	gripTime			   : TIME := T#250MS;                          // Време за ход на грипера
	gripTimeOut            : TIME := T#2S;                             // Време за отваряне/затваряне на гриперите
	insertTimeOut          : TIME := T#3S;                             // Време за движене нагоре/надолу на inserter 
    driveMoveTimeOut	   : TIME := T#4S;                             // Време за ход на мотора
	driveHomeTimeOut       : TIME := T#10S;                            // Време за home на мотора
	camTimeOut             : TIME := T#2S; 							   // Време за 1 снимка от камерата
	driveEnTime            : TIME := T#1S;                             // Време за ресет на инвертора на мотора
	drivePosTime           : TIME := T#100MS;                          // Време за задаване на задание за позициониране	

END_VAR


drivesControl();          // Упр. на ЛинМот мотора 

setStateVars(ioImage, activeState);


CASE activeState OF


//  *** Start Up
//  Старт на станцията след подаване на захр.	

	inserterLoadStates.stStartUp:
		setDisplayState(inserterLoadDisplayStates.dStStartUp);
		Stations.insertLoadDrive.DoEnable   := FALSE;
		Stations.insertLoadDrive.DoMove     := FALSE;	
		Stations.insertLoadDrive.DoHome     := FALSE;					   						   
		nextState(inserterLoadStates.stPowerUp);

//  *** Power Up - Start
//  Инициализация след подaване на захранване

	inserterLoadStates.stPowerUp:
		IF io.getSR(ioImage.xGrip_close, ioImage.xGrip_open) THEN
			setError(inserterLoadStates.stErrInitSensor);
		END_IF
		nextState(inserterLoadStates.stInit);

//  *** Init 
//  Инициализация на станцията
	
	inserterLoadStates.stInit:
	
		depWait(globalDeps.depILoadInitDone);		
		
		IF NOT resetDone THEN
			nextState(inserterLoadStates.stResetStart);
		END_IF
		
		IF prepareStart THEN
			nextState(inserterLoadStates.stPrepareStart);
		END_IF
		
		IF loadStart THEN
			nextState(inserterLoadStates.stLoadStart);
		END_IF		
		
		IF rotStart THEN
			nextState(inserterLoadStates.stRotStart);
		END_IF

		IF posStart THEN
			nextState(inserterLoadStates.stPosStart);
		END_IF

		IF insertStart THEN
			nextState(inserterLoadStates.stInsertStart);		
		END_IF	

		IF releaseStart THEN
			nextState(inserterLoadStates.stReleaseStart);
		END_IF	

		IF syncStart THEN
			nextState(inserterLoadStates.stSyncIndexStart);
		END_IF		
			
		nextState(inserterLoadStates.stInitDone);
		
// *** Init Done

	inserterLoadStates.stInitDone:
		nextState(inserterLoadStates.stReady);
	
// *** Ready

	inserterLoadStates.stReady:	
		setDisplayState(inserterLoadDisplayStates.dStStandBy);	
		IF Global.purgeDoneIL THEN
			resetDone          := FALSE;		
			Global.purgeDoneIL := FALSE;
		END_IF
		depNextState(Stations.machineStBase, GlobalDeps.depMachineStopping,  inserterLoadStates.stInserterLoadStopped);
		depNextState(Stations.machineStBase, GlobalDeps.depMachineStop,      inserterLoadStates.stInserterLoadStopped);	
		depWait(globalDeps.depILoadWaitIndex);
		nextState(inserterLoadStates.stPrepareStart);

// *** Inserter is Stopped

	inserterLoadStates.stInserterLoadStopped:
		setDisplayState(inserterLoadDisplayStates.dStStationIsStopped);	
		depWait(globalDeps.depILoadStop);
		depNextState(stations.machineStBase, GlobalDeps.depMachineAuto,       inserterLoadStates.stReady);
	    depNextState(Stations.machineStBase, GlobalDeps.depMachinePurgeStart, inserterLoadStates.stReady);			
		Stations.insertLoadDrive.DoEnable   := FALSE;
		Stations.insertLoadDrive.DoMove     := FALSE;	
		Stations.insertLoadDrive.DoHome     := FALSE;		

// *** Reset - Start
// Ресетиране на inserter

	inserterLoadStates.stResetStart:
		setDisplayState(inserterLoadDisplayStates.dStStationIsReseting);		
		resetDone := FALSE;		
		nextState(inserterLoadStates.stResetSyncRobot);
		
// *** Reset - Robot Sync
// Робота трябва да е на безопастно растояние

	inserterLoadStates.stResetSyncRobot:
		IF NOT GLobal.robotSafe THEN	
			depWait(globalDeps.depILoadWaitRobotReady);
			nextState(inserterLoadStates.stResetGripOpen);	
		ELSE
			nextState(inserterLoadStates.stResetGripOpen);	
		END_IF			

// *** Reset - Grip Open
// Отваряне на грипера

	inserterLoadStates.stResetGripOpen:
		io.setSR(ioImage.yGrip_open, ioImage.yGrip_close);
		nextState(inserterLoadStates.stResetGripCheck);	

// *** Reset - Grip Check
// Проверка дали грипера се е отворил
// Движение на гора на инсертъра

	inserterLoadStates.stResetGripCheck:		
 		IF io.getSR(ioImage.xGrip_open, ioImage.xGrip_close) THEN
			io.setSR(ioImage.yInsert_up, ioImage.yInsert_down);
			nextState(inserterLoadStates.stResetMoveUpCheck);	
		END_IF
		timeOutError(gripTimeOut, inserterLoadStates.stErrGripNotOpen);
		
// *** Reset - Move Up Check
// Проверка дали инсертъра е горе

	inserterLoadStates.stResetMoveUpCheck:		
		IF io.getSR(ioImage.xInsert_up, ioImage.xInsert_down) THEN
			nextState(inserterLoadStates.stResetLimitsCalc);			
		END_IF
		timeOutError(insertTimeOut, inserterLoadStates.stErrInsertNotUp);	
			
// *** Reset - Limit Check
// В зависимост от избраният модел на продукт се зараждат настойки в инвертора на мотора

	inserterLoadStates.stResetLimitsCalc:
			
		initRotPos    := Stations.insertLoadSetting.rotParams[Global.recipe].initRot;
		camRotPos     := Stations.insertLoadSetting.rotParams[Global.recipe].camRot;
		cwRotPos      := Stations.insertLoadSetting.rotParams[Global.recipe].cwRot;
		ccwRotPos     := Stations.insertLoadSetting.rotParams[Global.recipe].ccwRot;
		
		IF Stations.insertLoadDrive.Error THEN
			Stations.insertLoadDrive.DoReset  := TRUE;
		ELSE
			Stations.insertLoadDrive.DoReset  := FALSE;
			Stations.insertLoadDrive.DoEnable := TRUE;
			IF stateDelay(driveEnTime) THEN
				nextState(inserterLoadStates.stResetDriveHome);
			END_IF
		END_IF
		timeOutError(driveEnTime*2, inserterLoadStates.stErrDriveErr);
		
// *** Reset - Drive Home
// Рефериране на мотора

	inserterLoadStates.stResetDriveHome:		
		IF Stations.insertLoadDrive.Enabled AND NOT Stations.insertLoadDrive.Error THEN	
			Stations.insertLoadDrive.DoHome := TRUE;
			IF stateDelay(driveEnTime) THEN
				nextState(inserterLoadStates.stResetDriveCheck1);	
			END_IF
		ELSE
			setError(inserterLoadStates.stErrDriveErr);
	   END_IF	
		
// *** Reset - Drive Check
// Проверка дали реферирането на мотора е завършено

	inserterLoadStates.stResetDriveCheck1:		
		IF Stations.insertLoadDrive.Refferenced AND NOT Stations.insertLoadDrive.Error THEN
			Stations.insertLoadDrive.DoHome := FALSE;
			nextState(inserterLoadStates.stResetDriveMove);	
		END_IF
		timeOutError(driveHomeTimeOut, inserterLoadStates.stErrDriveHome);	

// *** Reset - Drive Move
// Ротатора застава на начална позиция

	inserterLoadStates.stResetDriveMove:
		IF Stations.insertLoadDrive.Enabled AND NOT Stations.insertLoadDrive.Error THEN	
			Stations.insertLoadDrive.TargetVelocity      := Stations.insertLoadSetting.axisWorkSpeed;
			Stations.insertLoadDrive.TargetAcceleration  := Stations.insertLoadSetting.axisAcc;
			Stations.insertLoadDrive.TargetPrecision     := Stations.insertLoadSetting.axisPres;
			Stations.insertLoadDrive.TargetPosition      := initRotPos;
		    Stations.insertLoadDrive.DoMove              := TRUE;
			IF stateDelay(driveEnTime) THEN			
				nextState(inserterLoadStates.stResetDriveCheck2);	
			END_IF
		ELSE
			setError(inserterLoadStates.stErrDriveErr);
	   END_IF	
	   
// *** Reset - Drive Check2
// Проверка дали реферирането на мотора е завършено

	inserterLoadStates.stResetDriveCheck2:		
		IF Stations.insertLoadDrive.TargetReached AND NOT Stations.insertLoadDrive.Error THEN
			Stations.insertLoadDrive.DoMove := FALSE;
			nextState(inserterLoadStates.stResetDone);	
		ELSIF NOT Stations.insertLoadDrive.TargetReached AND Stations.insertLoadDrive.Error THEN
			setError(inserterLoadStates.stErrDriveErr);
		END_IF	
		timeOutError(driveMoveTimeOut, inserterLoadStates.stErrDriveTimeOut);	

// *** Reset - Done

	inserterLoadStates.stResetDone:		
		resetDone := TRUE;
	    nextState(inserterLoadStates.stReady);			
		
// *** Prepare - Start
// Индекс масата е завършила ходата си - чака се робота да донесе сензор

	inserterLoadStates.stPrepareStart:
	   setDisplayState(inserterLoadDisplayStates.dStWorking);
	   prepareStart := TRUE;
	   nextState(inserterLoadStates.stPrepareNestCheck);	   
	   
// *** Prepare - Nest Check
// Ако в масата има зареден сенсор - станцията преключва работа
// Иначе дава сигнал на робота, че очаква от него да донесе сензор

	inserterLoadStates.stPrepareNestCheck:	   
		IF NOT io.getX(ioImage.xNest) AND NOT Global.purgeActive THEN
 	       nextState(inserterLoadStates.stPrepareRobotWait);  
        ELSE
	        prepareStart := FALSE;
 	        nextState(inserterLoadStates.stSyncIndexStart);  			
        END_IF	
	  
// *** Prepare - Robot Wait
// Изчаква робота да донесе сензор 

	inserterLoadStates.stPrepareRobotWait:		
		depSignal(globalDeps.depILoadSignalForLoad);
		depNextState(Stations.roboStBase, globalDeps.depRoboILoadOnPos, inserterLoadStates.stPrepareDone);
	
// *** Prepare - Done 

	inserterLoadStates.stPrepareDone:		
		prepareStart    := FALSE;
		nextState(inserterLoadStates.stLoadStart);
		
// *** Load - Start
// Сензора трябва да се прехвърли от робота в грипера на инсъртъра

	inserterLoadStates.stLoadStart:			
		loadStart   := TRUE;
		io.setSR(ioImage.yGrip_close, ioImage.yGrip_open);
		IF stateDelay(gripTime) THEN
			nextState(inserterLoadStates.stLoadGripCheck);	
		END_IF
	
// *** Load - Gripper Check
// Проверява се дали се е затворил грипера на инсъртъра

	inserterLoadStates.stLoadGripCheck:		
		IF io.getSR(ioImage.xGrip_close, ioImage.xGrip_open) THEN
			nextState(inserterLoadStates.stLoadRobotSync);	
		END_IF	
		timeOutError(gripTimeOut, inserterLoadStates.stErrGripNotClose);		
		
// *** Load - Robo Sync
// Дава се сигнал робота да си отвори грипера

	inserterLoadStates.stLoadRobotSync:			
		depWait(globalDeps.depRoboGripOpen);
		depNextState(Stations.roboStBase, GlobalDeps.depILoadRobotBack, inserterLoadStates.stLoadDone);

// *** Load - Done

	inserterLoadStates.stLoadDone:			
		loadStart  := FALSE;
		nextState(inserterLoadStates.stRotStart);		

// *** Rot - Start
// Започва ротиране на сензора, за да може да бъде сниман

	inserterLoadStates.stRotStart:	
		rotStart    := TRUE;
		io.setSR(ioImage.yGrip_close, ioImage.yGrip_open);
		nextState(inserterLoadStates.stRotGripCheck);

// *** Rot - Grip Check
// Ако е затворен грипера, пуска мотора 

	inserterLoadStates.stRotGripCheck:
		IF io.getSR(ioImage.xGrip_close, ioImage.xGrip_open) THEN
			IF Stations.insertLoadDrive.Enabled AND NOT Stations.insertLoadDrive.Error THEN
				nextState(inserterLoadStates.stRotDriveMove);	
			ELSE
			    nextState(inserterLoadStates.stRotDriveOn);			
			END_IF
		END_IF	
		timeOutError(gripTimeOut, inserterLoadStates.stErrGripNotClose);
		
// *** Rot - Drive On
// Ако е затворен грипера, пуска мотора 

	inserterLoadStates.stRotDriveOn:
		IF Stations.insertLoadDrive.Error THEN
			Stations.insertLoadDrive.DoReset  := TRUE;
		ELSE
			Stations.insertLoadDrive.DoReset  := FALSE;
			Stations.insertLoadDrive.DoEnable := TRUE;
			IF stateDelay(driveEnTime) THEN
				nextState(inserterLoadStates.stRotDriveMove);
			END_IF
		END_IF
		timeOutError(driveEnTime*2, inserterLoadStates.stErrDriveErr);

// *** Rot - Drive Move
// Завърта мотора на поз. за снимане

	inserterLoadStates.stRotDriveMove:
		IF Stations.insertLoadDrive.Enabled AND NOT Stations.insertLoadDrive.Error THEN	
			Stations.insertLoadDrive.TargetVelocity      := Stations.insertLoadSetting.axisWorkSpeed;
			Stations.insertLoadDrive.TargetAcceleration  := Stations.insertLoadSetting.axisAcc;
			Stations.insertLoadDrive.TargetPrecision     := Stations.insertLoadSetting.axisPres;
			Stations.insertLoadDrive.TargetPosition      := camRotPos;
		    Stations.insertLoadDrive.DoMove              := TRUE;	
			IF stateDelay(driveEnTime) THEN		
				nextState(inserterLoadStates.stRotDriveCheck);	
			END_IF
		ELSE
			setError(inserterLoadStates.stErrDriveErr);
	   END_IF	

// *** Rot - Drive Check
// Проверка дали мотора си е завършил хода

	inserterLoadStates.stRotDriveCheck:
		IF Stations.insertLoadDrive.TargetReached AND NOT Stations.insertLoadDrive.Error THEN
			Stations.insertLoadDrive.DoMove := FALSE;
			io.setY(ioImage.yFlashLight);
			nextState(inserterLoadStates.stRotCamShot);	
		ELSIF NOT Stations.insertLoadDrive.TargetReached AND Stations.insertLoadDrive.Error THEN
			setError(inserterLoadStates.stErrDriveErr);
		END_IF	
		timeOutError(driveMoveTimeOut, inserterLoadStates.stErrDriveTimeOut);

// *** Rot - Cam Shot
// Прави се снимка на сензора

	inserterLoadStates.stRotCamShot:
		Stations.insertLoadData := Global.recipe;
		nextState(inserterLoadStates.stRotCamCheck);

// *** Rot - Cam Check
// Проверява се дали има успешна снимка и върнат резултат

	inserterLoadStates.stRotCamCheck:
		IF Stations.insertLoadData = dataRequestCam.done THEN 
			io.rstY(ioImage.yFlashLight);
			
			IF TagsHMI.camResult <> camResult.null THEN
				
				CASE TagsHMI.camResult OF 
						camResult.turnCCW : workRotPos := ccwRotPos;
						camResult.turnCW  : workRotPos := cwRotPos;
				END_CASE
				nextState(inserterLoadStates.stRotDone);
				
			ELSE
				setError(inserterLoadStates.stErrCamBadResult);				
			END_IF
		
		ELSIF Stations.insertLoadData = dataRequestCam.error THEN
			setError(inserterLoadStates.stErrCamErr);			
		END_IF
		timeOutError(camTimeOut, inserterLoadStates.stErrCamTimeout);		
		
// *** Rot - Done

	inserterLoadStates.stRotDone:		
		rotStart   := FALSE;
		nextState(inserterLoadStates.stPosStart);		
		
// *** Pos  - Start
// Трябва да се завърти сензора на базата на резултата от камерата

	inserterLoadStates.stPosStart:		
		posStart   := TRUE;
		io.setSR(ioImage.yGrip_close, ioImage.yGrip_open);
		nextState(inserterLoadStates.stPosGripCheck);		
			
// *** Pos - Grip Check

	inserterLoadStates.stPosGripCheck:
		IF io.getSR(ioImage.xGrip_close, ioImage.xGrip_open) THEN
			IF Stations.insertLoadDrive.Enabled AND NOT Stations.insertLoadDrive.Error THEN
				nextState(inserterLoadStates.stPosDriveMove);	
			ELSE
			    nextState(inserterLoadStates.stPosDriveOn);			
			END_IF
		END_IF	
		timeOutError(gripTimeOut, inserterLoadStates.stErrGripNotClose);	
		
// *** Pos - Drive On
// Ако е затворен грипера, пуска мотора 

	inserterLoadStates.stPosDriveOn:
		IF Stations.insertLoadDrive.Error THEN
			Stations.insertLoadDrive.DoReset  := TRUE;
		ELSE
			Stations.insertLoadDrive.DoReset  := FALSE;
			Stations.insertLoadDrive.DoEnable := TRUE;
			IF stateDelay(driveEnTime) THEN
				nextState(inserterLoadStates.stPosDriveMove);
			END_IF
		END_IF
		timeOutError(driveEnTime*2, inserterLoadStates.stErrDriveErr);	
		
// *** Pos - Drive Move
// Завърта мотора 

	inserterLoadStates.stPosDriveMove:
		IF Stations.insertLoadDrive.Enabled AND NOT Stations.insertLoadDrive.Error THEN	
			Stations.insertLoadDrive.TargetVelocity      := Stations.insertLoadSetting.axisWorkSpeed;
			Stations.insertLoadDrive.TargetAcceleration  := Stations.insertLoadSetting.axisAcc;
			Stations.insertLoadDrive.TargetPrecision     := Stations.insertLoadSetting.axisPres;
			Stations.insertLoadDrive.TargetPosition      := workRotPos;
		    Stations.insertLoadDrive.DoMove              := TRUE;
			IF stateDelay(driveEnTime) THEN			
				nextState(inserterLoadStates.stPosDriveCheck);	
			END_IF
		ELSE
			setError(inserterLoadStates.stErrDriveErr);
	   END_IF	
		
// *** Pos - Drive Check
// Проверка дали мотора си е завършил хода

	inserterLoadStates.stPosDriveCheck:
		IF Stations.insertLoadDrive.TargetReached AND NOT Stations.insertLoadDrive.Error THEN
			Stations.insertLoadDrive.DoMove := FALSE;
			nextState(inserterLoadStates.stPosDone);	
		ELSIF NOT Stations.insertLoadDrive.TargetReached AND Stations.insertLoadDrive.Error THEN
			setError(inserterLoadStates.stErrDriveErr);
		END_IF	
		timeOutError(driveMoveTimeOut, inserterLoadStates.stErrDriveTimeOut);			   
	   
// *** Pos - Done

	inserterLoadStates.stPosDone:
		posStart   := FALSE;
		nextState(inserterLoadStates.stInsertStart);	  

// *** Insert - Start
// Поставя сензора на в гнездото на индекс масата

	inserterLoadStates.stInsertStart:
		insertStart := TRUE;
		io.setSR(ioImage.yGrip_close, ioImage.yGrip_open);
		nextState(inserterLoadStates.stInsertGripCheck);	

// *** Insert - Grip Check
// Проверява се дали грипера е затворен

	inserterLoadStates.stInsertGripCheck:
		IF io.getSR(ioImage.xGrip_close, ioImage.xGrip_open) THEN
			nextState(inserterLoadStates.stInsertNestCheck);		
		END_IF
		timeOutError(gripTimeOut, inserterLoadStates.stErrGripNotClose);
		
// *** Insert - Nest Check
// Сензор се поставя само ако на масата няма

	inserterLoadStates.stInsertNestCheck:
		IF NOT io.getX(ioImage.xNest) THEN
			io.setSR(ioImage.yInsert_down, ioImage.yInsert_up);
			nextState(inserterLoadStates.stInsertMoveDownCheck);			
		ELSE
			setError(inserterLoadStates.stErrInitSensor);
		END_IF
		
// *** Insert - Insert Move Down Check
// Проверява се дали е инсъртъра е долу

	inserterLoadStates.stInsertMoveDownCheck:		
		IF io.getSR(ioImage.xInsert_down, ioImage.xInsert_up) THEN
			nextState(inserterLoadStates.stInsetDone);			
		END_IF	
		timeOutError(insertTimeOut, inserterLoadStates.stErrInsertNotDown);

// *** Insert - Done

	inserterLoadStates.stInsetDone:	 
		insertStart := FALSE;
		nextState(inserterLoadStates.stReleaseStart);		
	   
// *** Release - Start
// Оставяне на сензора в гнездота и връщата в начална поз.

	inserterLoadStates.stReleaseStart:	   
		releaseStart := TRUE;
		io.setSR(ioImage.yGrip_open, ioImage.yGrip_close);
		nextState(inserterLoadStates.stReleaseGripCheck);	

// *** Release - Grip Check
// Проверка дали грипера се е отворил

	inserterLoadStates.stReleaseGripCheck:	   
		IF io.getSR(ioImage.xGrip_open, ioImage.xGrip_close) THEN
			io.setSR(ioImage.yInsert_up, ioImage.yInsert_down);
			nextState(inserterLoadStates.stReleaseMoveUpCheck);			
		END_IF	
		timeOutError(gripTimeOut, inserterLoadStates.stErrGripNotOpen);				   
	
// *** Release - Move Up Check
// Проверка дали инсъртъра е горе

	inserterLoadStates.stReleaseMoveUpCheck:
		IF io.getSR(ioImage.xInsert_up, ioImage.xInsert_down) THEN
			IF Stations.insertLoadDrive.Enabled AND NOT Stations.insertLoadDrive.Error THEN
				nextState(inserterLoadStates.stReleaseDriveMove);	
			ELSE
			    nextState(inserterLoadStates.stReleaseDriveOn);			
			END_IF			
		END_IF
		timeOutError(insertTimeOut, inserterLoadStates.stErrInsertNotUp);	

// *** Release - Drive On
// Ако инсъртъра е горе , пуска мотора 

	inserterLoadStates.stReleaseDriveOn:
		IF Stations.insertLoadDrive.Error THEN
			Stations.insertLoadDrive.DoReset  := TRUE;
		ELSE
			Stations.insertLoadDrive.DoReset  := FALSE;
			Stations.insertLoadDrive.DoEnable := TRUE;
			IF stateDelay(driveEnTime) THEN
				nextState(inserterLoadStates.stReleaseDriveMove);
			END_IF
		END_IF
		timeOutError(driveEnTime*2, inserterLoadStates.stErrDriveErr);	
		
// *** Release - Drive Move
// Завърта мотора 

	inserterLoadStates.stReleaseDriveMove:
		IF Stations.insertLoadDrive.Enabled AND NOT Stations.insertLoadDrive.Error THEN	
			Stations.insertLoadDrive.TargetVelocity      := Stations.insertLoadSetting.axisWorkSpeed;
			Stations.insertLoadDrive.TargetAcceleration  := Stations.insertLoadSetting.axisAcc;
			Stations.insertLoadDrive.TargetPrecision     := Stations.insertLoadSetting.axisPres;
			Stations.insertLoadDrive.TargetPosition      := initRotPos;
		    Stations.insertLoadDrive.DoMove              := TRUE;
			IF stateDelay(driveEnTime) THEN			
				nextState(inserterLoadStates.stReleaseDriveCheck);	
			END_IF
		ELSE
			setError(inserterLoadStates.stErrDriveErr);
	   END_IF	
		
// *** Release - Drive Check
// Проверка дали мотора си е завършил хода

	inserterLoadStates.stReleaseDriveCheck:
		IF Stations.insertLoadDrive.TargetReached AND NOT Stations.insertLoadDrive.Error THEN
			Stations.insertLoadDrive.DoMove := FALSE;
			nextState(inserterLoadStates.stReleaseDone);	
		ELSIF NOT Stations.insertLoadDrive.TargetReached AND Stations.insertLoadDrive.Error THEN
			setError(inserterLoadStates.stErrDriveErr);
		END_IF	
		timeOutError(driveMoveTimeOut, inserterLoadStates.stErrDriveTimeOut);  
	   
// *** Release - Done

	inserterLoadStates.stReleaseDone:	
        setDisplayState(inserterLoadDisplayStates.dStStationReady);	
		releaseStart  := FALSE;
		nextState(inserterLoadStates.stSyncIndexStart);

// *** Sync Index - Start
// Дава се разрешение да се завърти индекс масата

	inserterLoadStates.stSyncIndexStart:
		syncStart := TRUE;		
		depWait(globalDeps.depILoadDone);	
		depNextState(Stations.incCommStBase, globalDeps.depIncCycleDone, inserterLoadStates.stSyncIndexDone); 

// *** Sync Index - Done

	inserterLoadStates.stSyncIndexDone:
		syncStart := FALSE;
		nextState(inserterLoadStates.stReady);   
	        
// *** Step Block State
// В този state се влиза винаги след изпълняването на една стъпка при стъпков режим
	inserterLoadStates.stStepBlock:
        setDisplayState(inserterLoadDisplayStates.dStWaitForNextStep);	
		
// *** Station Stop
// Станцията е била изключена 
 
	inserterLoadStates.stStop: 	
		Stations.insertLoadDrive.DoEnable   := FALSE;
		Stations.insertLoadDrive.DoMove     := FALSE;	
	    resetDone			                := FALSE; 						   
	    prepareStart                        := FALSE; 						   
	    loadStart                           := FALSE; 						   
	    rotStart                            := FALSE; 						   
	    posStart                            := FALSE; 						   
	    insertStart                         := FALSE;							  
	    releaseStart                        := FALSE; 						   
	    syncStart			                := FALSE; 

// *** ERROR - Grip Not Open
// Грипера не се е отворил на време

	inserterLoadStates.stErrGripNotOpen:
		setDisplayState(inserterLoadDisplayStates.dStGripperDidNotOpen); 

// *** ERROR - Grip Not Close
// Грипера не се е затворил на време

	inserterLoadStates.stErrGripNotClose:
		setDisplayState(inserterLoadDisplayStates.dStGripperDidNotClose);
		
// *** ERROR - Inserter Not Down
// Inserter не е стинглал долна позиция на време

	inserterLoadStates.stErrInsertNotDown:
		setDisplayState(inserterLoadDisplayStates.dStInserterDidNotMoveDown);		
		
// *** ERROR - Inserter Not Up
// Inserter не е стинглал горна позиция на време

	inserterLoadStates.stErrInsertNotUp:
		setDisplayState(inserterLoadDisplayStates.dStInserterDidNotMoveUp);		
		
// *** ERROR - Drive Homming TimeOut
// ЛинМот мотора не е могъл да се homming както трябва

	inserterLoadStates.stErrDriveHome:
		setDisplayState(inserterLoadDisplayStates.dStDriveDidNotHome);
		Stations.insertLoadDrive.DoEnable   := FALSE;
		Stations.insertLoadDrive.DoMove     := FALSE;	
		Stations.insertLoadDrive.DoHome     := FALSE;	
		
// *** ERROR - Drive Homming TimeOut
// ЛинМот инвертора е върнал грешка

	inserterLoadStates.stErrDriveErr:
		setDisplayState(inserterLoadDisplayStates.dStDriveError);	
		Stations.insertLoadDrive.DoEnable   := FALSE;
		Stations.insertLoadDrive.DoMove     := FALSE;		
		
// *** ERROR - Drive Move TimeOut
// ЛинМот мотора не е завършил движението си навреме

	inserterLoadStates.stErrDriveTimeOut:
		setDisplayState(inserterLoadDisplayStates.dStDriveTimeOutMove);	
		Stations.insertLoadDrive.DoEnable   := FALSE;
		Stations.insertLoadDrive.DoMove     := FALSE;		
		
// *** ERROR - Camera Timeout
// Камерата се е забавила твърде мн. с връщането на резултат

	inserterLoadStates.stErrCamTimeout:
		setDisplayState(inserterLoadDisplayStates.dStCameraTimeOut);
		
// *** ERROR - Camera Error
// Камерата се е забавила твърде мн. с връщането на резултат

	inserterLoadStates.stErrCamErr:
		setDisplayState(inserterLoadDisplayStates.dStCameraError);
		
// *** ERROR - Camera Error
// Камерата е върнала грешен резултат

	inserterLoadStates.stErrCamBadResult:
		setDisplayState(inserterLoadDisplayStates.dStCameraBadResult);	
		
	
// *** ERROR - Init sensor 
// При старт на машаината не може да има захванат от грипера сензор

	inserterLoadStates.stErrInitSensor:	
		setDisplayState(inserterLoadDisplayStates.dStInitSensorGripError);	
		
// *** EMG Stop
// Аварийно спиране при натискане на гъба или отваряне на врата

	inserterLoadStates.stEMG:		
		Stations.insertLoadDrive.DoEnable   := FALSE;
		Stations.insertLoadDrive.DoMove     := FALSE;	
		Stations.insertLoadDrive.DoHome     := FALSE;
		nextState(inserterLoadStates.stInit);		


END_CASE

ACTION drivesControl:


axisLinMot       ( TargetPosition 		   := Stations.insertLoadDrive.TargetPosition,
				   TargetVelocity 		   := Stations.insertLoadDrive.TargetVelocity,
				   TargetAcceleration	   := Stations.insertLoadDrive.TargetAcceleration,
				   TargetDeceleration	   := Stations.insertLoadDrive.TargetAcceleration,
				   TargetPrecision 		   := Stations.insertLoadDrive.TargetPrecision,			
				   IsAbsolute 			   := FALSE,
	               OperationMode		   := Stations.insertLoadDrive.OperationMode,     				
	               Enabled 				   => Stations.insertLoadDrive.Enabled,
	               Error 				   => Stations.insertLoadDrive.Error,
	               ErrorID 				   => Stations.insertLoadDrive.ErrorID,
	               Refferenced 			   => Stations.insertLoadDrive.Refferenced,
	               Moving 				   => Stations.insertLoadDrive.Moving,
	               CurrentPosition 		   => Stations.insertLoadDrive.CurrentPosition,
	               CurrentVelocity		   => Stations.insertLoadDrive.CurrentVelocity,             				
				   Axis					   := Stations.insertLoadAxis,
		           DoServoOn 			   := Stations.insertLoadDrive.DoEnable, 
	               DoHome 				   := Stations.insertLoadDrive.DoHome, 
	               DoMove 				   := Stations.insertLoadDrive.DoMove, 
	               DoReset 				   := Stations.insertLoadDrive.DoReset, 
	               TargetReached 		   := Stations.insertLoadDrive.TargetReached, 
	               DoStop 				   := Stations.insertLoadDrive.DoStop);
END_ACTION

END_FUNCTION_BLOCK

// ---- POUs/Stations/insertUnloadStation.TcPOU
FUNCTION_BLOCK insertUnloadStation EXTENDS stateMachine
VAR_INPUT
	
	ioImage                : inserterUnloadImage;

END_VAR

VAR

	activeState            : inserterUnloadStates;	
	axisLinMot             : FB_ServoAxis_LinMot; 
	
	resetDone			   : BOOL := FALSE; 						   // Инсъртъра е ресетнат
	prepareStart           : BOOL := FALSE; 						   // Ако има сенсор в гнездото, завърта грипера 
	moveDownStart          : BOOL := FALSE; 						   // Слиза да вземе сензора
	unloadSensorStart      : BOOL := FALSE; 						   // Взима сензора и инсъртъра се вдига нагоре
	posStart               : BOOL := FALSE; 						   // Ротира грипера за взимане на сензора от робота
	releaseStart           : BOOL := FALSE; 						   // Подава сензора на робота
	syncRobot              : BOOL := false;                            // Робота е на безопастно място
	syncStart			   : BOOL := FALSE; 						   // Sync с индекс масата, че работа е завършена
	
	
	initRotPos			   : REAL; 									   // Начално завъртане
	workRotPos             : REAL;                                     // Завъртане за може робота да вземе сензора
	
	gripTime			   : TIME := T#250MS;                          // Време за ход на грипера                                     
	gripTimeOut            : TIME := T#2S;                             // Време за отваряне/затваряне на гриперите
	insertTimeOut          : TIME := T#3S;                             // Време за движене нагоре/надолу на inserter
    driveMoveTimeOut	   : TIME := T#4S;                             // Време за ход на мотора
	driveHomeTimeOut       : TIME := T#10S;                            // Време за home на мотора
	sensorTime             : TIME := T#250MS; 						   // Време за за реакция на лазерен сензор
	driveEnTime            : TIME := T#1S;                             // Време за ресет на инвертора на мотора
	drivePosTime           : TIME := T#100MS;                          // Време за задаване на задание за позициониране	

END_VAR


drivesControl();          // Упр. на ЛинМот мотора 

setStateVars(ioImage, activeState);

CASE activeState OF
	

//  *** Start Up
//  Старт на станцията след подаване на захр.	

	inserterUnloadStates.stStartUp:
		setDisplayState(inserterUnLoadDisplayStates.dStStartUp);
		Stations.insertUnLoadDrive.DoEnable   := FALSE;
		Stations.insertUnLoadDrive.DoMove     := FALSE;	
		Stations.insertUnLoadDrive.DoHome     := FALSE;					   						   
		nextState(inserterUnloadStates.stPowerUp);

//  *** Power Up - Start
//  Инициализация след подaване на захранване

	inserterUnloadStates.stPowerUp:
		IF io.getSR(ioImage.xGrip_close, ioImage.xGrip_open) THEN
			setError(inserterUnloadStates.stErrInitSensor);
		END_IF
		nextState(inserterUnloadStates.stInit);

//  *** Init 
//  Инициализация на станцията
	
	inserterUnloadStates.stInit:
	
		depWait(globalDeps.depULoadInitDone);	
		
		IF NOT resetDone THEN
			nextState(inserterUnloadStates.stResetStart);
		END_IF
		
		IF prepareStart THEN
			nextState(inserterUnloadStates.stPrepareStart);
		END_IF
		
		IF moveDownStart THEN
			nextState(inserterUnloadStates.stMoveDownStart);
		END_IF		
		
		IF unloadSensorStart THEN
			nextState(inserterUnloadStates.stUnloadSensorStart);
		END_IF

		IF posStart THEN
			nextState(inserterUnloadStates.stPosStart);
		END_IF

		IF releaseStart THEN
			nextState(inserterUnloadStates.stReleaseStart);
		END_IF	
		
		IF syncRobot THEN
			nextState(inserterUnloadStates.stReleaseDone);
		END_IF

		IF syncStart THEN
			nextState(inserterUnloadStates.stSyncIndexStart);
		END_IF		
			
		nextState(inserterUnloadStates.stInitDone);
		
// *** Init Done

	inserterUnloadStates.stInitDone:
		nextState(inserterUnloadStates.stReady);
	
// *** Ready

	inserterUnloadStates.stReady:	
		setDisplayState(inserterUnLoadDisplayStates.dStStandBy);	
		IF Global.purgeDoneIU THEN
			resetDone          := FALSE;		
			Global.purgeDoneIU := FALSE;
		END_IF
		depNextState(Stations.machineStBase, GlobalDeps.depMachineStopping,  inserterUnloadStates.stInserterUnloadStopped);
		depNextState(Stations.machineStBase, GlobalDeps.depMachineStop,      inserterUnloadStates.stInserterUnloadStopped);	
		depWait(globalDeps.depULoadWaitIndex);
		nextState(inserterUnloadStates.stPrepareStart);

// *** Inserter is Stopped

	inserterUnloadStates.stInserterUnloadStopped:
		setDisplayState(inserterUnLoadDisplayStates.dStStationIsStopped);
		depWait(globalDeps.depULoadStop);
		depNextState(stations.machineStBase, GlobalDeps.depMachineAuto,       inserterUnloadStates.stReady);
	    depNextState(Stations.machineStBase, GlobalDeps.depMachinePurgeStart, inserterUnloadStates.stReady);			
		Stations.insertUnLoadDrive.DoEnable   := FALSE;
		Stations.insertUnLoadDrive.DoMove     := FALSE;	
		Stations.insertUnLoadDrive.DoHome     := FALSE;

// *** Reset - Start
// Ресетиране на inserter

	inserterUnloadStates.stResetStart:
		setDisplayState(inserterUnLoadDisplayStates.dStStationIsReseting);	
		resetDone := FALSE;		
		nextState(inserterUnloadStates.stResetSyncRobot);
		
// *** Reset - Robot Sync
// Робота трябва да е на безопастно растояние

	inserterUnloadStates.stResetSyncRobot:
		IF NOT Global.robotSafe THEN	
			depWait(globalDeps.depULoadWaitRobotReady);
			nextState(inserterUnloadStates.stResetGripOpen);	
	    ELSE
			nextState(inserterUnloadStates.stResetGripOpen);
		END_IF		

// *** Reset - Grip Open
// Отваряне на грипера

	inserterUnloadStates.stResetGripOpen:
		io.setSR(ioImage.yGrip_open, ioImage.yGrip_close);
		nextState(inserterUnloadStates.stResetGripCheck);	

// *** Reset - Grip Check
// Проверка дали грипера се е отворил.
// Движение на гора на инсертъра

	inserterUnloadStates.stResetGripCheck:		
 		IF io.getSR(ioImage.xGrip_open, ioImage.xGrip_close) THEN
			io.setSR(ioImage.yInsert_up, ioImage.yInsert_down);
			nextState(inserterUnloadStates.stResetMoveUpCheck);	
		END_IF
		timeOutError(gripTimeOut, inserterUnloadStates.stErrGripNotOpen);
		
// *** Reset - Move Up Check
// Проверка дали инсертъра е горе

	inserterUnloadStates.stResetMoveUpCheck:		
		IF io.getSR(ioImage.xInsert_up, ioImage.xInsert_down) THEN
			nextState(inserterUnloadStates.stResetLimitsCalc);			
		END_IF
		timeOutError(insertTimeOut, inserterUnloadStates.stErrInsertNotUp);	
			
// *** Reset - Limit Check
// В зависимост от избраният модел на продукт се зараждат настойки в инвертора на мотора

	inserterUnloadStates.stResetLimitsCalc:
			
		initRotPos     := Stations.insertUnloadSetting.rotParams[Global.recipe].initRot;
		workRotPos     := Stations.insertUnloadSetting.rotParams[Global.recipe].workRot;

		
		IF Stations.insertUnLoadDrive.Error THEN
			Stations.insertUnLoadDrive.DoReset  := TRUE;
		ELSE
			Stations.insertUnLoadDrive.DoReset  := FALSE;
			Stations.insertUnLoadDrive.DoEnable := TRUE;
			IF stateDelay(driveEnTime) THEN
				nextState(inserterUnloadStates.stResetDriveHome);
			END_IF
		END_IF
		timeOutError(driveEnTime*2, inserterUnloadStates.stErrDriveErr);
		
// *** Reset - Drive Home
// Рефериране на мотора

	inserterUnloadStates.stResetDriveHome:		
		IF Stations.insertUnLoadDrive.Enabled AND NOT Stations.insertUnLoadDrive.Error THEN	
			Stations.insertUnLoadDrive.DoHome := TRUE;
			IF stateDelay(drivePosTime) THEN
				nextState(inserterUnloadStates.stResetDriveCheck);	
			END_IF	
		ELSE
			setError(inserterUnloadStates.stErrDriveErr);
	   END_IF	
		
// *** Reset - Drive Check
// Проверка дали реферирането на мотора е завършено

	inserterUnloadStates.stResetDriveCheck:		
		IF Stations.insertUnLoadDrive.Refferenced AND NOT Stations.insertUnLoadDrive.Error THEN
			Stations.insertUnLoadDrive.DoHome := FALSE;
			nextState(inserterUnloadStates.stResetDone);	
		END_IF
		timeOutError(driveHomeTimeOut, inserterUnloadStates.stErrDriveHome);	

// *** Reset - Done

	inserterUnloadStates.stResetDone:		
		resetDone := TRUE;
	    nextState(inserterUnloadStates.stReady);		
		
// *** Prepare - Start
// Индекс масата е завършила ходата си 

	inserterUnloadStates.stPrepareStart:
       setDisplayState(inserterUnLoadDisplayStates.dStWorking);	 
	   prepareStart := TRUE;
	   io.setSR(ioImage.yGrip_open, ioImage.yGrip_close);
	   io.setSR(ioImage.yInsert_up, ioImage.yInsert_down);
	   nextState(inserterUnloadStates.stPrepareGripCheck);		
		
// *** Prepare - Grip Check
// Инсертера трябва да е горе и грипера му да е отворен

	inserterUnloadStates.stPrepareGripCheck:		
		IF io.getSR(ioImage.xGrip_open, ioImage.xGrip_close) AND 
		   io.getSR(ioImage.xInsert_up, ioImage.xInsert_down) THEN
				nextState(inserterUnloadStates.stPrepareNestCheck);
		ELSE
			IF stateDelay(insertTimeOut) THEN
				IF NOT io.getSR(ioImage.xGrip_open, ioImage.xGrip_close) THEN
					setError(inserterUnloadStates.stErrGripNotOpen);
				ELSIF io.getSR(ioImage.xInsert_up, ioImage.xInsert_down) THEN
					setError(inserterUnloadStates.stErrInsertNotUp);
				END_IF
			END_IF
		END_IF	
				
// *** Prepare - Nest Check
// За да започне цикъла на станицята, трябва да има в сензор в гнездото
// и InC да е върнало, че този сензор е със статус GOOD

	inserterUnloadStates.stPrepareNestCheck:	
		IF stateDelay(sensorTime) THEN
			IF io.getX(ioImage.xNest) AND Global.sensorStatus THEN
				Global.sensorOnIUnload := TRUE; 			
				IF Stations.insertUnloadDrive.Enabled AND NOT Stations.insertUnloadDrive.Error THEN
					nextState(inserterUnloadStates.stPrepareDriveMove);
				ELSE
					nextState(inserterUnloadStates.stPrepareDriveOn);
				END_IF
			ELSIF io.getX(ioImage.xNest) XOR GLobal.sensorStatus THEN
				setError(inserterUnloadStates.stErrNestSensor);
			ELSE	
				prepareStart := FALSE;
				nextState(inserterUnloadStates.stSyncIndexStart);
			END_IF
		END_IF	

// *** Prepare - Drive On
// Захранване на мотора ако не е пуснат 

	inserterUnloadStates.stPrepareDriveOn:
		IF Stations.insertUnLoadDrive.Error THEN
			Stations.insertUnLoadDrive.DoReset  := TRUE;
		ELSE
			Stations.insertUnLoadDrive.DoReset  := FALSE;
			Stations.insertUnLoadDrive.DoEnable := TRUE;
			IF stateDelay(driveEnTime) THEN
				nextState(inserterUnloadStates.stPrepareDriveMove);
			END_IF
		END_IF
		timeOutError(driveEnTime*2, inserterUnloadStates.stErrDriveErr);

// *** Prepare - Drive Move
// Завърта мотора на поз. за изваждането на сензор

	inserterUnloadStates.stPrepareDriveMove:
		IF Stations.insertUnLoadDrive.Enabled AND NOT Stations.insertUnLoadDrive.Error THEN	
			Stations.insertUnLoadDrive.TargetVelocity      := Stations.insertUnLoadSetting.axisWorkSpeed;
			Stations.insertUnLoadDrive.TargetAcceleration  := Stations.insertUnLoadSetting.axisAcc;
			Stations.insertUnLoadDrive.TargetPrecision     := Stations.insertUnLoadSetting.axisPres;
			Stations.insertUnLoadDrive.TargetPosition      := initRotPos;
		    Stations.insertUnLoadDrive.DoMove              := TRUE;	
			IF stateDelay(drivePosTime) THEN		
				nextState(inserterUnloadStates.stPrepareDriveCheck);	
			END_IF	
		ELSE
			setError(inserterUnloadStates.stErrDriveErr);
	   END_IF	

// *** Prepare - Drive Check
// Проверка дали мотора си е завършил хода

	inserterUnloadStates.stPrepareDriveCheck:
		IF Stations.insertUnLoadDrive.TargetReached AND NOT Stations.insertUnLoadDrive.Error THEN
			Stations.insertUnLoadDrive.DoMove := FALSE;
			nextState(inserterUnloadStates.stPrepareDone);	
		ELSIF NOT Stations.insertUnLoadDrive.TargetReached AND Stations.insertUnLoadDrive.Error THEN
			setError(inserterUnloadStates.stErrDriveErr);
		END_IF	
		timeOutError(driveMoveTimeOut, inserterUnloadStates.stErrDriveTimeOut);

// *** Prepare - Done

	inserterUnloadStates.stPrepareDone:		
		prepareStart := FALSE;
	    nextState(inserterUnloadStates.stMoveDownStart);		
		
// *** Move Down  - Start
// Инсертера слиза надолу зада вземе сензор от гнездото на масата

	inserterUnloadStates.stMoveDownStart:	 
	   moveDownStart := TRUE;
	   io.setSR(ioImage.yGrip_open, ioImage.yGrip_close);
	   io.setSR(ioImage.yInsert_up, ioImage.yInsert_down);
	   nextState(inserterUnloadStates.stMoveDownGripCheck);	
		
// *** Move Down - Grip Check
// Инсертера трябва да е горе и грипера му да е отворен

	inserterUnloadStates.stMoveDownGripCheck:		
		IF io.getSR(ioImage.xGrip_open, ioImage.xGrip_close) AND 
		   io.getSR(ioImage.xInsert_up, ioImage.xInsert_down) THEN
		   		io.setSR(ioImage.yInsert_down, ioImage.yInsert_up);
				nextState(inserterUnloadStates.stMoveDownCheck);
		ELSE
			IF stateDelay(insertTimeOut) THEN
				IF NOT io.getSR(ioImage.xGrip_open, ioImage.xGrip_close) THEN
					setError(inserterUnloadStates.stErrGripNotOpen);
				ELSIF io.getSR(ioImage.xInsert_up, ioImage.xInsert_down) THEN
					setError(inserterUnloadStates.stErrInsertNotUp);
				END_IF
			END_IF
		END_IF			
		
// *** Move Down - Down Check
// Инсертера трябва да е долу

	inserterUnloadStates.stMoveDownCheck:		
		IF io.getSR(ioImage.xInsert_down, ioImage.xInsert_up) THEN
			nextState(inserterUnloadStates.stMoveDownDone);
		END_IF
		timeOutError(insertTimeOut, inserterUnloadStates.stErrInsertNotDown);	
		
// *** Move Down - Done

	inserterUnloadStates.stMoveDownDone:		
		moveDownStart := FALSE;
	    nextState(inserterUnloadStates.stUnloadSensorStart);		

// *** Unload Sensor - Start
// Грипера се затваря, захваща сензора и го изважда от гнездото на масата

	inserterUnloadStates.stUnloadSensorStart:	
		unloadSensorStart := TRUE;
		io.setSR(ioImage.yGrip_open, ioImage.yGrip_close);
		io.setSR(ioImage.yInsert_down, ioImage.yInsert_up);
	    nextState(inserterUnloadStates.stUnloadSensorGripCheck1);			

// *** Unload Sensor - Grip Check 1
// Проверка на гриперите

	inserterUnloadStates.stUnloadSensorGripCheck1:
		IF io.getSR(ioImage.xGrip_open, ioImage.xGrip_close) AND 
		   io.getSR(ioImage.xInsert_down, ioImage.xInsert_up) THEN
		   		io.setSR(ioImage.yGrip_close, ioImage.yGrip_open);
				nextState(inserterUnloadStates.stUnloadSensorGripCheck2);
		ELSE
			IF stateDelay(insertTimeOut) THEN
				IF NOT io.getSR(ioImage.xGrip_open, ioImage.xGrip_close) THEN
					setError(inserterUnloadStates.stErrGripNotOpen);
				ELSIF io.getSR(ioImage.xInsert_down, ioImage.xInsert_up) THEN
					setError(inserterUnloadStates.stErrInsertNotDown);
				END_IF
			END_IF
		END_IF	

// *** Unload Sensor - Grip Check 2
// Проверка  дали грипера се е затворил 

	inserterUnloadStates.stUnloadSensorGripCheck2:
		IF io.getSR(ioImage.xGrip_close, ioImage.xGrip_open) AND stateDelay(gripTime) THEN
			io.setSR(ioImage.yInsert_up, ioImage.yInsert_down);
			nextState(inserterUnloadStates.stUnloadSensorMoveCheck);
		END_IF	
		timeOutError(gripTimeOut, inserterUnloadStates.stErrGripNotClose);			
	
// *** Unload Sensor - Move Check
// Проверка  дали инсертера е горе

	inserterUnloadStates.stUnloadSensorMoveCheck:
		IF io.getSR(ioImage.xInsert_up, ioImage.xInsert_down) THEN
			nextState(inserterUnloadStates.stUnloadSensorDone);
		END_IF	
		timeOutError(insertTimeOut, inserterUnloadStates.stErrInsertNotUp);

// *** Unload Sensor - Done

	inserterUnloadStates.stUnloadSensorDone:		
		unloadSensorStart := FALSE;
	    nextState(inserterUnloadStates.stPosStart);
		
// *** Pos - Start
// Сензора трябва да се ротира, че да може да го хване робота

	inserterUnloadStates.stPosStart:
		posStart := TRUE;
		io.setSR(ioImage.yGrip_close, ioImage.yGrip_open);
		io.setSR(ioImage.yInsert_up, ioImage.yInsert_down);
		nextState(inserterUnloadStates.stPosGripCheck);

// *** Pos - Grip Check

	inserterUnloadStates.stPosGripCheck:		
		IF io.getSR(ioImage.xGrip_close, ioImage.xGrip_open) AND 
		   io.getSR(ioImage.xInsert_up, ioImage.xInsert_down) THEN
				IF Stations.insertUnloadDrive.Enabled AND NOT Stations.insertUnloadDrive.Error THEN
					nextState(inserterUnloadStates.stPosDriveMove);
				ELSE
					nextState(inserterUnloadStates.stPosDriveOn);
				END_IF
		ELSE
			IF stateDelay(insertTimeOut) THEN
				IF NOT io.getSR(ioImage.xGrip_close, ioImage.xGrip_open) THEN
					setError(inserterUnloadStates.stErrGripNotClose);
				ELSIF io.getSR(ioImage.xInsert_up, ioImage.xInsert_down) THEN
					setError(inserterUnloadStates.stErrInsertNotUp);
				END_IF
			END_IF
		END_IF			
		
// *** Pos - Drive On
// Захранване на мотора ако не е пуснат 

	inserterUnloadStates.stPosDriveOn:
		IF Stations.insertUnLoadDrive.Error THEN
			Stations.insertUnLoadDrive.DoReset  := TRUE;
		ELSE
			Stations.insertUnLoadDrive.DoReset  := FALSE;
			Stations.insertUnLoadDrive.DoEnable := TRUE;
			IF stateDelay(driveEnTime) THEN
				nextState(inserterUnloadStates.stPosDriveMove);
			END_IF
		END_IF
		timeOutError(driveEnTime*2, inserterUnloadStates.stErrDriveErr);

// *** Pos - Drive Move
// Завърта мотора на поз. за взимане на сензора от робота

	inserterUnloadStates.stPosDriveMove:
		IF Stations.insertUnLoadDrive.Enabled AND NOT Stations.insertUnLoadDrive.Error THEN	
			Stations.insertUnLoadDrive.TargetVelocity      := Stations.insertUnLoadSetting.axisWorkSpeed;
			Stations.insertUnLoadDrive.TargetAcceleration  := Stations.insertUnLoadSetting.axisAcc;
			Stations.insertUnLoadDrive.TargetPrecision     := Stations.insertUnLoadSetting.axisPres;
			Stations.insertUnLoadDrive.TargetPosition      := workRotPos;
		    Stations.insertUnLoadDrive.DoMove              := TRUE;	
			IF stateDelay(drivePosTime) THEN		
				nextState(inserterUnloadStates.stPosDriveCheck);
			END_IF	
		ELSE
			setError(inserterUnloadStates.stErrDriveErr);
	   END_IF	
		
// *** Pos - Drive Check
// Проверка дали мотора си е завършил хода

	inserterUnloadStates.stPosDriveCheck:
		IF Stations.insertUnLoadDrive.TargetReached AND NOT Stations.insertUnLoadDrive.Error THEN
			Stations.insertUnLoadDrive.DoMove := FALSE;
			nextState(inserterUnloadStates.stPosDone);	
		ELSIF NOT Stations.insertUnLoadDrive.TargetReached AND Stations.insertUnLoadDrive.Error THEN
			setError(inserterUnloadStates.stErrDriveErr);
		END_IF	
		timeOutError(driveMoveTimeOut, inserterUnloadStates.stErrDriveTimeOut);		
		
// *** Pos - Done

	inserterUnloadStates.stPosDone:		
		posStart := FALSE;
		nextState(inserterUnloadStates.stReleaseStart);
		
// *** Release - Start
// Робота взима сензора от инсъртъра

	inserterUnloadStates.stReleaseStart:		
		releaseStart := TRUE;		
		nextState(inserterUnloadStates.stReleaseSyncRobot);		
		
// *** Release - Sync Robot
// Изчаква се робота 

	inserterUnloadStates.stReleaseSyncRobot:		
		depSync(Stations.roboStBase, globalDeps.depRoboULoadOnPos);
		depNextState(Stations.roboStBase, globalDeps.depRoboGripClose, inserterUnloadStates.stReleaseGripOpen);	
		
// *** Release - Grip Open
// Отваря грипера

	inserterUnloadStates.stReleaseGripOpen:	
		io.setSR(ioImage.yGrip_open, ioImage.yGrip_close);
		nextState(inserterUnloadStates.stReleaseGripCheck);		
		
// *** Release - Grip Check
// Проверка дали грипера е отворен

	inserterUnloadStates.stReleaseGripCheck:
		IF io.getSR(ioImage.xGrip_open, ioImage.xGrip_close) THEN
			nextState(inserterUnloadStates.stReleaseLoadDone);				
		END_IF
		timeOutError(gripTimeOut, inserterUnloadStates.stErrGripNotOpen);			
		
// *** Release - Load Done
// Грипера се е отворил и сензора е захванат успешно от робота

	inserterUnloadStates.stReleaseLoadDone:	
		setDisplayState(inserterUnLoadDisplayStates.dStStationReady);
		depWait(globalDeps.depRoboLoadSensor);	
		nextState(inserterUnloadStates.stReleaseDone);

// *** Release - Done

	inserterUnloadStates.stReleaseDone:	
		releaseStart := FALSE;
		syncRobot    := TRUE;
		depSync(Stations.roboStBase, globalDeps.depULoadRobotOutOfRich);
		nextState(inserterUnloadStates.stSyncIndexStart);	
		
// *** Sync Index - Start
// Дава се разрешение да се завърти индекс масата

	inserterUnloadStates.stSyncIndexStart:
		syncStart := TRUE;		
		syncRObot := FALSE;
		depWait(globalDeps.depULoadDone);	
		depNextState(Stations.incCommStBase, globalDeps.depIncCycleDone, inserterUnloadStates.stSyncIndexDone);

// *** Sync Index - Done

	inserterUnloadStates.stSyncIndexDone:
		syncStart := FALSE;
		nextState(inserterUnloadStates.stReady);		
	
	   
// *** Step Block State
// В този state се влиза винаги след изпълняването на една стъпка при стъпков режим
	inserterUnloadStates.stStepBlock:
		setDisplayState(inserterUnLoadDisplayStates.dStWaitForNextStep);
		
// *** Station Stop
// Станцията е била изключена 
 
	inserterUnloadStates.stStop: 	
		Stations.insertUnLoadDrive.DoEnable   := FALSE;
		Stations.insertUnLoadDrive.DoMove     := FALSE;	
		resetDone			  				  := FALSE; 						   
		prepareStart          				  := FALSE; 						   
		moveDownStart          				  := FALSE; 						   
		unloadSensorStart     				  := FALSE; 						  
		posStart                			  := FALSE; 						   
		releaseStart           				  := FALSE; 						   
		syncRobot              				  := FALSE;                            
		syncStart			    			  := FALSE; 						   	

// *** ERROR - Grip Not Open
// Грипера не се е отворил на време

	inserterUnloadStates.stErrGripNotOpen:
		setDisplayState(inserterUnloadDisplayStates.dStGripperDidNotOpen); 

// *** ERROR - Grip Not Close
// Грипера не се е затворил на време

	inserterUnloadStates.stErrGripNotClose:
		setDisplayState(inserterUnloadDisplayStates.dStGripperDidNotClose);
		
// *** ERROR - Inserter Not Down
// Inserter не е стинглал долна позиция на време

	inserterUnloadStates.stErrInsertNotDown:
		setDisplayState(inserterUnloadDisplayStates.dStInserterDidNotMoveDown);		
		
// *** ERROR - Inserter Not Up
// Inserter не е стинглал горна позиция на време

	inserterUnloadStates.stErrInsertNotUp:
		setDisplayState(inserterUnloadDisplayStates.dStInserterDidNotMoveUp);		
		
// *** ERROR - Drive Homming TimeOut
// ЛинМот мотора не е могъл да се homming както трябва

	inserterUnloadStates.stErrDriveHome:
		setDisplayState(inserterUnloadDisplayStates.dStDriveDidNotHome);
		Stations.insertUnLoadDrive.DoEnable   := FALSE;
		Stations.insertUnLoadDrive.DoMove     := FALSE;	
		Stations.insertUnLoadDrive.DoHome     := FALSE;	
		
// *** ERROR - Drive Homming TimeOut
// ЛинМот инвертора е върнал грешка

	inserterUnloadStates.stErrDriveErr:
		setDisplayState(inserterUnloadDisplayStates.dStDriveError);	
		Stations.insertUnLoadDrive.DoEnable   := FALSE;
		Stations.insertUnLoadDrive.DoMove     := FALSE;		
		
// *** ERROR - Drive Move TimeOut
// ЛинМот мотора не е завършил движението си навреме

	inserterUnloadStates.stErrDriveTimeOut:
		setDisplayState(inserterUnloadDisplayStates.dStDriveTimeOutMove);	
		Stations.insertUnLoadDrive.DoEnable   := FALSE;
		Stations.insertUnLoadDrive.DoMove     := FALSE;		
					
// *** ERROR - Init sensor 
// При старт на машаината не може да има захванат от грипера сензор

	inserterUnloadStates.stErrInitSensor:	
		setDisplayState(inserterUnloadDisplayStates.dStInitSensorGripError);

// *** ERROR - No Nest Sensor 
// InC е върнало сигнал че има сенсор в гнездото, но лазера не отчита нищо там

	inserterUnloadStates.stErrNestSensor:	
		setDisplayState(inserterUnloadDisplayStates.dStNoSensorInNest);	
		
// *** EMG 
// Аварийно спиране при натискане на гъба или отваряне на врата

	inserterUnloadStates.stEMG:		
		Stations.insertUnLoadDrive.DoEnable   := FALSE;
		Stations.insertUnLoadDrive.DoMove     := FALSE;	
		Stations.insertUnLoadDrive.DoHome     := FALSE;
		nextState(inserterUnloadStates.stInit);	

END_CASE

ACTION drivesControl:


axisLinMot       ( TargetPosition 		   := Stations.insertUnloadDrive.TargetPosition,
				   TargetVelocity 		   := Stations.insertUnloadDrive.TargetVelocity,
				   TargetAcceleration	   := Stations.insertUnloadDrive.TargetAcceleration,
				   TargetDeceleration	   := Stations.insertUnloadDrive.TargetAcceleration,
				   TargetPrecision 		   := Stations.insertUnloadDrive.TargetPrecision,			
				   IsAbsolute 			   := FALSE,
	               OperationMode		   := Stations.insertUnloadDrive.OperationMode,     				
	               Enabled 				   => Stations.insertUnloadDrive.Enabled,
	               Error 				   => Stations.insertUnloadDrive.Error,
	               ErrorID 				   => Stations.insertUnloadDrive.ErrorID,
	               Refferenced 			   => Stations.insertUnloadDrive.Refferenced,
	               Moving 				   => Stations.insertUnloadDrive.Moving,
	               CurrentPosition 		   => Stations.insertUnloadDrive.CurrentPosition,
	               CurrentVelocity		   => Stations.insertUnloadDrive.CurrentVelocity,             				
				   Axis					   := Stations.insertUnLoadAxis,
		           DoServoOn 			   := Stations.insertUnloadDrive.DoEnable, 
	               DoHome 				   := Stations.insertUnloadDrive.DoHome, 
	               DoMove 				   := Stations.insertUnloadDrive.DoMove, 
	               DoReset 				   := Stations.insertUnloadDrive.DoReset, 
	               TargetReached 		   := Stations.insertUnloadDrive.TargetReached, 
	               DoStop 				   := Stations.insertUnloadDrive.DoStop);
END_ACTION

END_FUNCTION_BLOCK

// ---- POUs/Stations/roboArmStation.TcPOU
FUNCTION_BLOCK roboArmStation EXTENDS stateMachine
VAR_INPUT
	
	ioImage                : roboArmImage;

END_VAR

VAR

	activeState            : roboArmStates;	
	
	initDone			   : BOOL := FALSE; 						   // Робота е инизиализиран
	resetActive            : BOOL := FALSE;                            // Процедура за homming  на робота - ипълнявасе за повечето движение след EMG или Err
	nextMoveStart          : BOOL := FALSE;                            // Тук се решава следващият ход на робота
	moveToEmptyStart       : BOOL := FALSE;                            // Робота отива да вземе тара от чакащата поз.
	emptyToUnloadStart     : BOOL := FALSE;                            // Тара се мести от чакащата поз. на изходен стакер
	unloadPalletStart      : BOOL := FALSE;                            // Робота подава празна тара на изх. стакер за закл.
	loadPalletStart        : BOOL := FALSE;                            // Има празна тара за взимане от вх. стакер
	emptyPosStart          : BOOL := FALSE;                            // Робота премества празна тара на чакащата поз.
	loadStart              : BOOL := FALSE;                            // Робота търси сензор за взимане от входната тара
	unloadStart            : BOOL := FALSE;                            // Робота търси място да остави сензор в изх. тара
	lInsertStart           : BOOL := FALSE;                            // Робота трябва да зареди със сензор Load Inserter
	lInsertLockStart       : BOOL := FALSE;                            // Подаване на сензора от робота към Load Inserter
	lInsertBack            : BOOL := FALSE;                            // Зареждането на сензора в Load Inserter е завършено
	uInsertStart           : BOOL := FALSE;                            // Робота трябва да вземе сензора от Unload Inserter
	uInsertLockStart       : BOOL := FALSE;                            // Взимане на сензора от робота към Uload Inserter
	uInsertBack            : BOOL := FALSE;                            // Вимането на сензора в Load Inserter е завършено	
	
	fixturesCount          : INT; 									   // Брой гнезда на тара спрямо избраната рецепта
	loadFixtures           : INT; 									   // Брой гнезда на входната тара
	unLoadFixtures         : INT; 									   // Брой гнезда на изходната тара
	typeHEX24              : BOOL;                                     // Работи се с HEX 24 
	typeHEX27              : BOOL;                                     // Работи се с HEX 27 	
    lamp24On               : BOOL;                                     // Сигнализация че оператора трябва да постави празна тара на чакаща поз. HEX24                              
	lamp27On               : BOOL;                                     // Сигнализация че оператора трябва да постави празна тара на чакаща поз. HEX27 
	palletIn			   : BOOL := FALSE;                            // Има захваната празна тара от робота
	palletMiss             : BOOL;                                     // На чакаща поз. липсва тара - робота не е донесъл
	palletOnEmptyPos       : BOOL;                                     // На чакаща поз. има поставена тара
	purgeActive            : BOOL;                                     // Има активна процедура PURGE
	initWaitLStacker       : BOOL;
	tempUnloadMove         : BOOL;
	checkLoadStacker       : BOOL;
	blockRunForLoad        : BOOL;	                                   // Изх. втакер е празен - робота на мръдва, докато не се заредят нови тари
	waitPosPalletRot       : DINT := 0;
	palletRotTypeWaitPos   : DINT;

	
	xWaitPos               : REFERENCE TO imageIO;                     // В зависимост от рецептата се използва само едната чакаща поз. 
	xSlideUp               : REFERENCE TO imageIO;
	xSLideDown             : REFERENCE TO imageIO;
    ySlideUp			   : REFERENCE TO imageIO;
	ySlideDown             : REFERENCE TO imageIO;
	yPalletLoadGrip        : REFERENCE TO imageIO;
	yPalletLoadFree        : REFERENCE TO imageIO;
  
	
	TON_0				   : TON;                                      // Тимери за мигането на лампите за чакащата поз.
	TON_1                  : TON;
	TOF_0                  : TOF;
	TOF_1                  : TOF;	
	
	gripTime			   : TIME := T#250MS;                          // Време за ход на грипера  	
	gripTimeOut            : TIME := T#2S;                             // Време за отваряне/затваряне на гриперите
	rotTimeOut             : TIME := T#2S;                             // Време за завъртане на сензора	
	slideTime              : TIME := T#2S;                             // Време за сваляне/качване на слайдера за тара
	palletGripTime         : TIME := T#500MS;                          // Време за захващатане на тара от "мекия" грипер
	robotHomeTime          : TIME := T#45S;                            // Време за ресетване на робота - изпълнение на HOME
	robotMoveTime		   : TIME := T#10S;                            // Макс. време за ход на робота
	robotResetTime         : TIME := T#1S;                             // Време за рестарт на робота
	sensorTime             : TIME := T#250MS;                          // Време за отчитане на сигнал от лазерната ролетка
	rotAfterTime		   : TIME := T#500MS;                             // След ход на робота, след това време за обръща сензора
	

END_VAR


signalLamps(enable   := palletOnEmptyPos,
			lamp24   := lamp24On, 
			sensor24 :=	io.getX(ioImage.xWaitPos24),		
            lamp27   := lamp27On, 
			sensor27 :=	io.getX(ioImage.xWaitPos27) );

setStateVars(ioImage, activeState);


CASE activeState OF 
	

// *** Starting Up
//  Старт на станцията след подаване на захр.
	
	roboArmStates.stStartUp:
		setDisplayState(roboArmDisplayStates.dStPowerUp);
		nextState(roboArmStates.stPowerUp);
		
// *** Power Up
// Проверява се дали няма останал сензор в робота

	roboArmStates.stPowerUp:
		IF io.getSR(ioImage.xGrip_close, ioImage.xGrip_open) THEN
			setError(roboArmStates.stErrInitSensor);
		END_IF
		
		IF io.getX(ioImage.xWaitPos24) THEN
			setError(roboArmStates.stErrInitPalletOn24);
		END_IF
		
		IF io.getX(ioImage.xWaitPos27) THEN
			setError(roboArmStates.stErrInitPalletOn27);
		END_IF		
	
// *** Init 
//  Инициализация на станцията

	roboArmStates.stInit:
		IF blockRunForLoad THEN
			IF NOT Global.lStackLastPallet THEN
				blockRunForLoad := FALSE;
			END_IF
		ELSE
			depWait(globalDeps.depRoboInitDone);
			IF TagsRobot.robotError THEN
				nextState(roboArmStates.stRobotReset);	
			ELSE 
				Stations.roboData := dataRequestRobot.done;
				nextState(roboArmStates.stRobotResetDone);
			END_IF
		END_IF
			
		
// *** Robot Reset 
//  Ресерване на грешката в робота

	roboArmStates.stRobotReset:
		Stations.roboData := dataRequestRobot.roboInit;
		nextState(roboArmStates.stRobotResetDone);		

// *** Robot Reset Done

	roboArmStates.stRobotResetDone:
		IF Stations.roboData = dataRequestRobot.done THEN
			IF resetActive THEN
				nextState(roboArmStates.stResetStart);
			ELSE
				nextState(roboArmStates.stNextRobotState);	
			END_IF							
		END_IF
		IF Stations.roboData = dataRequestRobot.error THEN
			nextState(roboArmStates.stErrRobot);
		END_IF
		timeOutError(robotResetTime, roboArmStates.stErrRobotTimeOut);
		
// *** Next Robot State
		
	roboArmStates.stNextRobotState:
	
		IF initWaitLStacker THEN
			nextState(roboArmStates.stInitWaitLoadStacker);			
		END_IF

		IF NOT initDone THEN
			nextState(roboArmStates.stInitStart);
		END_IF

		IF nextMoveStart THEN
			nextState(roboArmStates.stNextMoveStart);
		END_IF	

		IF moveToEmptyStart THEN
			nextState(roboArmStates.stMoveToEmptyStart);
		END_IF	
	
		IF emptyToUnloadStart THEN
			nextState(roboArmStates.stEmptyToUnloadMove);
		END_IF
		
		IF unloadPalletStart THEN
			nextState(roboArmStates.stUnloadPalletStart);
		END_IF	
		
		IF loadPalletStart THEN
			nextState(roboArmStates.stLoadPalletStart);
		END_IF	
		
		IF emptyPosStart THEN
			nextState(roboArmStates.stEmptyPosStart);
		END_IF		
		
		IF loadStart THEN
			nextState(roboArmStates.stLoadStart);
		END_IF		
		
		IF unloadStart THEN
			nextState(roboArmStates.stUnloadStart);
		END_IF	
		
		IF lInsertStart THEN
			nextState(roboArmStates.stLInsertStart);
		END_IF	

		IF lInsertLockStart THEN
			nextState(roboArmStates.stLInsertLockStart);
		END_IF	
		
		IF lInsertBack THEN
			nextState(roboArmStates.stLInsertBackStart);
		END_IF	

		IF uInsertStart THEN
			nextState(roboArmStates.stUInsertStart);
		END_IF		
		
		IF uInsertLockStart THEN
			nextState(roboArmStates.stUInsertLockStart);
		END_IF		
		
		IF uInsertBack THEN
			nextState(roboArmStates.stUInsertBackStart);
		END_IF				
		
		nextState(roboArmStates.stInitDone);	
	
// *** Init Done	
	
	roboArmStates.stInitDone:
		nextState(roboArmStates.stReady);
 
// *** Ready

	roboArmStates.stReady:
		setDisplayState(roboArmDisplayStates.dStWorking);	
		depNextState(Stations.machineStBase,  globalDeps.depMachineStopping,  roboArmStates.stStationStop);
		depNextState(Stations.machineStBase,  globalDeps.depMachineStop,      roboArmStates.stStationStop);
		IF purgeActive THEN
			nextState(roboArmStates.stPurgeStart);			
		END_IF
		nextState(roboArmStates.stNextMoveStart);		

// *** Station Stop	
	
	roboArmStates.stStationStop:
		setDisplayState(roboArmDisplayStates.dStPowerUp);
		depWait(globalDeps.depRoboStop);
		depNextState(stations.machineStBase, globalDeps.depMachineAuto, 	  roboArmStates.stInit);
		depNextState(stations.machineStBase, globalDeps.depMachinePurgeStart, roboArmStates.stPurgeStart);
		Global.robotSafe := TRUE;

// *** Purge  - Start	
	
	roboArmStates.stPurgeStart:
		purgeActive      := TRUE;	
		Global.robotSafe := FALSE;		
		depNextState(stations.machineStBase, globalDeps.depMachinePurgeRobot,  roboArmStates.stPurgeMove);	
		IF Global.sensorOnIUnload THEN
			nextState(roboArmStates.stUInsertStart);		
		END_IF
		
// *** Purge - Move
// Премества се робота на HOME поз.	
	
	roboArmStates.stPurgeMove:
		Stations.roboData := dataRequestRobot.roboPrg_Home;
		nextState(roboArmStates.stPurgeMoveCheck);	
		
// *** Purge - Move Check
// Робота изпчълни ли си хода ?
	
	roboArmStates.stPurgeMoveCheck:
		IF Stations.roboData = dataRequestRobot.done THEN
			nextState(roboArmStates.stPurgeSync);
		END_IF
		IF Stations.roboData = dataRequestRobot.error THEN
			nextState(roboArmStates.stErrRobot);
		END_IF
		timeOutError(robotHomeTime, roboArmStates.stErrRobotReset);
		
// *** Purge - Sync 
	
	roboArmStates.stPurgeSync:		
		depWait(globalDeps.depRoboPurgeDone); 
		nextState(roboArmStates.stPurgeMoveDone);			
			
// *** Purge - Done 
	
	roboArmStates.stPurgeMoveDone:
		purgeActive := FALSE;
		initDone    := FALSE; 
		nextState(roboArmStates.stStationStop);	

// *** Init - Start
// Робота се прибира на безопасно място и инициялизира тулинга си

	roboArmStates.stInitStart:
		initDone          := FALSE;
		resetActive       := FALSE;
        Stations.roboData := dataRequestRobot.done;		
		nextState(roboArmStates.stInitMoveHome);
		
// *** Init - Move Home
// Задаване на робота програма HOME

	roboArmStates.stInitMoveHome:
		Stations.roboData := dataRequestRobot.roboPrg_Home;
		nextState(roboArmStates.stInitMoveCheck);
		
// *** Init - Move Check
// Проверка дали се е робота е на HOME поз.

	roboArmStates.stInitMoveCheck:
		IF Stations.roboData = dataRequestRobot.done THEN
			io.setSR(ioImage.yGrip_open, ioImage.yGrip_close);
			io.setSR(ioImage.yRot_home, ioImage.yRot_back);
			io.setSR(ioImage.ySlide24_up, ioImage.ySlide24_down);
			io.setSR(ioImage.ySlide27_up, ioImage.ySlide27_down);
			nextState(roboArmStates.stInitToolCheck);
		END_IF
		IF Stations.roboData = dataRequestRobot.error THEN
			nextState(roboArmStates.stErrRobot);
		END_IF
		timeOutError(robotHomeTime, roboArmStates.stErrRobotReset);

// *** Init - Tool Check
// Проверка дали толинга на робота се е инциализирал

	roboArmStates.stInitToolCheck:
		IF io.getSR(ioImage.xGrip_open, ioImage.xGrip_close) AND
		   io.getSR(ioImage.xRot_home, ioImage.xRot_back)    AND
		   io.getSR(ioImage.xSlide24_up, ioImage.xSlide24_down) AND
		   io.getSR(ioImage.xSlide27_up, ioImage.xSlide27_down)  THEN
		   		nextState(roboArmStates.stInitLoadRecipe);
		END_IF
		
		IF stateDelay(slideTime * 2) THEN
			IF NOT io.getSR(ioImage.xGrip_open, ioImage.xGrip_close) THEN
				setError(roboArmStates.stErrGripNotOpen);
			END_IF
		
			IF NOT io.getSR(ioImage.xRot_home, ioImage.xRot_back) THEN
				setError(roboArmStates.stErrRotNotTurn0);
			END_IF

			IF NOT io.getSR(ioImage.xSlide24_up, ioImage.xSlide24_down) OR
			   NOT io.getSR(ioImage.xSlide27_up, ioImage.xSlide27_down)THEN
				setError(roboArmStates.stErrSlideNotUp);
			END_IF
		END_IF	

// *** Init - Load Recipe
// Заражда правилната рецепта в зависимост от подадените данни от InC

	roboArmStates.stInitLoadRecipe:
		fixturesCount := Stations.roboSetings.roboArmParams[Global.recipe].fixtureNum;		
		IF Stations.roboSetings.roboArmParams[Global.recipe].waitPos24 THEN
			xWaitPos 		 REF= ioImage.xWaitPos24;
			xSlideUp 		 REF= ioImage.xSlide24_up;
			xSlideDown       REF= ioImage.xSlide24_down;
			ySlideUp         REF= ioImage.ySlide24_up;
			ySlideDown       REF= ioImage.ySlide24_down;
			yPalletLoadGrip  REF= ioImage.yPalletLoad24;
			yPalletLoadFree  REF= ioImage.yPalletLoad27;    //  така работи 24, да не се обръща
			typeHEX24 := TRUE; 
			typeHEX27 := FALSE;			
		ELSIF Stations.roboSetings.roboArmParams[Global.recipe].waitPos27 THEN
			xWaitPos 		 REF= ioImage.xWaitPos27;
			xSlideUp 		 REF= ioImage.xSlide27_up;
			xSlideDown       REF= ioImage.xSlide27_down;
			ySlideUp         REF= ioImage.ySlide27_up;
			ySlideDown       REF= ioImage.ySlide27_down;
			yPalletLoadGrip  REF= ioImage.yPalletLoad27;
			yPalletLoadFree  REF= ioImage.yPalletLoad24;    //  така работи 27, да не се обръща
			typeHEX27 := TRUE;
			typeHEX24 := FALSE;  			
		END_IF	
		io.setSR(yPalletLoadFree, yPalletLoadGrip);
		palletOnEmptyPos        := TRUE;		
		TagsRobot.roboRecipeNum := Global.recipe;
		nextState(roboArmStates.stInitRecipeCheck);		

// *** Init - Recipe Check
// Проверка дали е заредена рецептата в робота

	roboArmStates.stInitRecipeCheck:
		IF Stations.roboData = dataRequestRobot.done THEN
			nextState(roboArmStates.stInitSyncStations);
		END_IF	
		IF Stations.roboData = dataRequestRobot.error THEN
			nextState(roboArmStates.stErrRobot);
		END_IF
		timeOutError(robotMoveTime, roboArmStates.stErrRobot);

// *** Init - Sync Stations
// Робота се е ресетнал - сега могат да се движат и останали станций

	roboArmStates.stInitSyncStations:
		IF NOT Global.robotSafe THEN
			depSync(Stations.sLoadStBase,        globalDeps.depSLoadWaitRobotReady);		
			depSync(Stations.sUnloadStBase,      globalDeps.depSUnloadWaitRobotReady);		
			depSync(Stations.insertLoadStBase,   globalDeps.depILoadWaitRobotReady);		
			depSync(Stations.insertUnloadStBase, globalDeps.depULoadWaitRobotReady);
			nextState(roboArmStates.stInitWaitLoadStacker);	
		ELSE
			nextState(roboArmStates.stInitWaitLoadStacker);	
		END_IF					


// *** Init - Wait Load Stacker
// Изчакава вх. стакер да си зареди тарите
// Тук се влиза след EMG -  оператора трябва да отвори вратите да зареди тари
// Сиглилзира на другите станций, че робота е на безопастно място - не е направено добре
// С глобална променлиеа - порази факта, че има само едно dependancy за state !

	roboArmStates.stInitWaitLoadStacker:
		initWaitLStacker := TRUE;	
		Global.robotSafe := TRUE;	
    	depWait(globalDeps.depSLoadStationReady);	
		nextState(roboArmStates.stInitReady);		
	
// *** Init - Ready

	roboArmStates.stInitReady:	
		initDone           := TRUE;
		initWaitLStacker   := FALSE;
		Global.robotSafe   := FALSE;
    	loadFixtures       := fixturesCount;
		Global.emptyLoadPallet    := FALSE;
		nextState(roboArmStates.stMoveToEmptyStart);	
		
// *** Reset - Start
// Робота се прибира на Home позицията си и в зависимост дали е взел сенсор или тара
// се избира следващият state

	roboArmStates.stResetStart:	
		resetActive := TRUE;
		nextState(roboArmStates.stResetSlider);		
	
// *** Reset - Slider
// Ако няма захваната тара робота вдига слайдера нагора 
// Ako има захваната тара грипера за тарата и слайдера не се пипат

	roboArmStates.stResetSlider:	
		IF 	palletIn THEN
			nextState(roboArmStates.stResetGrip);	
		ELSE
			io.setSR(yPalletLoadFree, yPalletLoadGrip);
			IF stateDelay(palletGripTime) THEN
				io.setSR(ySlideUp, ySlideDown);
			    nextState(roboArmStates.stResetSliderCheck);				
			END_IF
		END_IF
	
// *** Reset - Slider Check
// Няма захваната тара и се проверява дали слайдера е горе

	roboArmStates.stResetSliderCheck:	
		IF io.getSR(xSlideUp, xSlideDown) THEN 
			nextState(roboArmStates.stResetGrip);
		END_IF
		timeOutError(slideTime, roboArmStates.stErrSlideNotUp);	

// *** Reset - Grip
// Ако има сензор в грипера на робота той не се пипа
// Ако няма може грипера да се отвори

	roboArmStates.stResetGrip:
		IF io.getSR(ioImage.xGrip_close, ioImage.xGrip_open) THEN
			Stations.roboData := dataRequestRobot.roboPrg_Home;	
			nextState(roboArmStates.stResetMoveCheck);			
		ELSE
			io.setSR(ioImage.yGrip_open, ioImage.xGrip_close);
			nextState(roboArmStates.stResetGripCheck);	
		END_IF	

// *** Reset - Grip Check
// В грипера на робота е нямало сензор 
// Проверява се дали се е отворил

	roboArmStates.stResetGripCheck:
		IF io.getSR(ioImage.xGrip_open, ioImage.xGrip_close) THEN
			Stations.roboData := dataRequestRobot.roboPrg_Home;	
			nextState(roboArmStates.stResetMoveCheck);				
		END_IF
		timeOutError(gripTimeOut, roboArmStates.stErrGripNotOpen);	

// *** Reset - Move Check
// Проверка дали робота е в HOME

	roboArmStates.stResetMoveCheck:
		IF Stations.roboData = dataRequestRobot.done THEN
			io.setSR(ioImage.yRot_home, ioImage.yRot_back);
			nextState(roboArmStates.stResetRotCheck);
		END_IF	
		IF Stations.roboData = dataRequestRobot.error THEN
			nextState(roboArmStates.stErrRobot);
		END_IF
		timeOutError(robotHomeTime, roboArmStates.stErrRobotReset);

// *** Reset - Rot Check
// Проверка дали ротатора се е завъртял на 0 град.

	roboArmStates.stResetRotCheck:
		IF io.getSR(ioImage.xRot_home, ioImage.xRot_back) THEN
			nextState(roboArmStates.stResetSync);				
		END_IF
		timeOutError(rotTimeOut, roboArmStates.stErrRotNotTurn0);	
		
// *** Reset - Sync
// Синхронизазия с останалите станция, че робота е готов

	roboArmStates.stResetSync:	
		nextState(roboArmStates.stNextRobotState);				

// *** Reset - Done

	roboArmStates.stResetDone:
		resetActive := FALSE;
		nextState(roboArmStates.stInit);

// *** Next Move - Start
// Тук се рещава какъв е следващият ход на робота на базата на ред условия

	roboArmStates.stNextMoveStart:
        nextMoveStart := TRUE;
        resetActive   := TRUE;
		IF checkLoadStacker AND loadFixtures = 0 THEN
			depWait(globalDeps.depSLoadStationReady);
		   	nextState(roboArmStates.stNextMoveWaitLStacker);	
		ELSE
			nextState(roboArmStates.stNextMovePalletCheck);
		END_IF	
		
// *** Next Move  - Wait Load Stacker
// Изчаква се вх. стакер да си свърши работата

	roboArmStates.stNextMoveWaitLStacker:
		checkLoadStacker := FALSE;		
		loadFixtures     := fixturesCount;
		Global.emptyLoadPallet  := FALSE;
		nextState(roboArmStates.stNextMovePalletCheck);	

// *** Next Move - Pallet Check
// Ако робота има захванта тара, то:
// 1. Има бройки на изх. тара - захванатата тара се оставя на чакащата поз.
// 2. Няма борйки на изх. тара захванатата тара се мести на изх. стакер

	roboArmStates.stNextMovePalletCheck:
		checkLoadStacker := FALSE;
		IF palletIn THEN
			IF unLoadFixtures > 0 OR Global.lStackLastPallet THEN
				nextMoveStart := FALSE;
				nextState(roboArmStates.stEmptyPosStart);				
			ELSE
				IF NOT tempUnloadMove THEN
					depSync(Stations.sUnloadStBase, globalDeps.depSUnloadStationReady);
					nextState(roboArmStates.stNextMoveSync);
				ELSE
					nextState(roboArmStates.stNextMoveSync);
				END_IF
				END_IF							
			END_IF
		nextState(roboArmStates.stNextMoveUnlodeFull);	

//*** Next MOVE - Sync
// ИЗходния стакер трява да е готов 

	roboArmStates.stNextMoveSync:	
	tempUnloadMove := TRUE;
 	Stations.roboData := dataRequestRobot.roboPrg_HomeWithPallet;
	nextState(roboArmStates.stNextMovePalletHome);

//*** Next MOVE - Sync
// ИЗходния стакер трява да е готов 

	roboArmStates.stNextMovePalletHome:	
		IF Stations.roboData = dataRequestRobot.done THEN	
 	        Stations.roboData := dataRequestRobot.roboPrg_UnloadStacker;			
			nextState(roboArmStates.stNextMoveCheck1);
		END_IF		
		IF Stations.roboData = dataRequestRobot.error THEN
			nextState(roboArmStates.stErrRobot);
		END_IF
		timeOutError(robotMoveTime, roboArmStates.stErrRobotTimeOut);	
		
// *** Next Move - Move Check
// Робота е занесъл празна тара над изх. стакер ?

	roboArmStates.stNextMoveCheck1:	
		IF Stations.roboData = dataRequestRobot.done THEN			
			nextState(roboArmStates.stNextMovePass);
		END_IF		
		IF Stations.roboData = dataRequestRobot.error THEN
			nextState(roboArmStates.stErrRobot);
		END_IF
		timeOutError(robotMoveTime, roboArmStates.stErrRobotTimeOut);			

// *** Next Move - Pass 1 

	roboArmStates.stNextMovePass:
	    tempUnloadMove := FALSE;
		nextMoveStart  := FALSE;	
		nextState(roboArmStates.stUnloadPalletStart);
		
// *** Next Move - Unload Full
// Изх. тара е пълна и трябва да се смени:
// 1. Ако има тара на чакаща поз. - тя се взима
// 2. Ако вх. тарата е празна     - тя се взима 

	roboArmStates.stNextMoveUnlodeFull:
	
		IF unLoadFixtures = 0 THEN		
		
			IF palletOnEmptyPos THEN
				IF io.getX(xWaitPos) THEN 
			    	Stations.roboData   := dataRequestRobot.roboPrg_EmptyPlace;	
					nextState(roboArmStates.stNextMoveEmptyCheck);	
				ELSE									// На чакащата поз. е трябвало да има тара, но няма !
					IF typeHEX24 THEN
						lamp24On := TRUE;
						lamp27On := FALSE;
					ELSIF typeHEX27 THEN
						lamp24On := FALSE;
						lamp27On := TRUE;
					END_IF	
					setError(roboArmStates.stErrNoPalletWaitPos);
				END_IF		
		
			ELSIF NOT palletOnEmptyPos AND loadFixtures = 0 THEN
				nextState(roboArmStates.stNextMoveLoadMove);	
			END_IF	
		
		END_IF
		nextState(roboArmStates.stNextMoveLoadEmpty);		

// *** Next Move - EmptyCheck
// Робота трябва да е над чакащата поз. 

	roboArmStates.stNextMoveEmptyCheck:
		IF Stations.roboData = dataRequestRobot.done THEN
			depSignal(globalDeps.depRoboUnLodPalletFull);
			nextState(roboArmStates.stNextMovePalletOnUload);
		END_IF		
		IF Stations.roboData = dataRequestRobot.error THEN
			nextState(roboArmStates.stErrRobot);
		END_IF
		timeOutError(robotMoveTime, roboArmStates.stErrRobotTimeOut);	
	
// *** Next Move - EmptyCheck
// Тарата може да се захване от робота

	roboArmStates.stNextMovePalletOnUload:
		nextMoveStart := FALSE;	
		nextState(roboArmStates.stMoveToEmptySliderDown);

// *** Next Move - Load 
// Робота отива над вх. стакер

	roboArmStates.stNextMoveLoadMove:		
		Stations.roboData   := dataRequestRobot.roboPrg_LoadStacker;	
		nextState(roboArmStates.stNextMoveLoadMoveCheck);			

// *** Next Move - Load Check
// Робота трябва да е над вх. стакер

	roboArmStates.stNextMoveLoadMoveCheck:		
		IF Stations.roboData = dataRequestRobot.done THEN	
			depSignal(globalDeps.depRoboUnLodPalletFull);		
			nextState(roboArmStates.stNextMoveLoadDone);	
		END_IF	
		IF Stations.roboData = dataRequestRobot.error THEN
			nextState(roboArmStates.stErrRobot);
		END_IF
		timeOutError(robotMoveTime, roboArmStates.stErrRobotTimeOut);

// *** Next Move - Load Done
// Изх. стакер може да заради тара 

	roboArmStates.stNextMoveLoadDone:	
			nextMoveStart := FALSE;			
			nextState(roboArmStates.stLoadPalletStart);			
		
// *** Next Move - Load Empty
// Входната тара е празна трябв да се зенесе на чакаща поз.
// Тук на изх. тара все още има място 

	roboArmStates.stNextMoveLoadEmpty:		
		IF loadFixtures = 0 AND unLoadFixtures > 0 THEN	
			IF NOT io.getX(xWaitPos) THEN
				Stations.roboData := dataRequestRobot.roboPrg_LoadStacker;				
				nextState(roboArmStates.stNextMoveCheck2);	
			ELSE 
				setError(roboArmStates.stErrPalletOnWaitPos);
			END_IF		
		END_IF
		nextState(roboArmStates.stNextNewCycle);			
			
// *** Next Move - Load Empty
// Робота трябва да е над вх. стакер

	roboArmStates.stNextMoveCheck2:		
		IF Stations.roboData = dataRequestRobot.done THEN			
			nextMoveStart := FALSE;			
			nextState(roboArmStates.stLoadPalletStart);	
		END_IF	
		IF Stations.roboData = dataRequestRobot.error THEN
			nextState(roboArmStates.stErrRobot);
		END_IF
		timeOutError(robotMoveTime, roboArmStates.stErrRobotTimeOut);			
			
// *** Next Move - New Cycle
// Във вх. тара има сензор
// Във изх. тара има още място - робота продължава

	roboArmStates.stNextNewCycle:	
		IF loadFixtures > 0 AND unLoadFixtures > 0 THEN
			nextMoveStart := FALSE;			
			nextState(roboArmStates.stLoadStart);	
		ELSE
			// изх. стакер е празен, вх. е пълен и е няма тара на чакаща пoз.
			// затова се кара оператора да сложи тари на чакащата поз.
			palletOnEmptyPos := TRUE;
			IF typeHEX24 THEN
				lamp24On := TRUE;
				lamp27On := FALSE;
		    ELSIF typeHEX27 THEN
				lamp24On := FALSE;
				lamp27On := TRUE;
			END_IF	
			nextState(roboArmStates.stNextMoveUnlodeFull);		
		END_IF

// *** Move to Empty - Start
// Празна тара се взиама от чакащата поз. и се премества отгоре на изходният стакер

	roboArmStates.stMoveToEmptyStart:
		moveToEmptyStart   := TRUE;	
		resetActive        := TRUE;
		nextState(roboArmStates.stMoveToEmptyCheck);		
		
// *** Move to Empty - Check
// На чакаща поз. трябва да има тара
// Ако има робота отива там 

	roboArmStates.stMoveToEmptyCheck:		
		IF io.getX(xWaitPos) THEN
			lamp24On 		   := FALSE;
			lamp27On           := FALSE;	
		    Stations.roboData  := dataRequestRobot.roboPrg_EmptyPlace;
			nextState(roboArmStates.stMoveToEmptyMoveCheck);	
		ELSE
			IF typeHEX24 THEN
				lamp24On := TRUE;
				lamp27On := FALSE;
			ELSIF typeHEX27 THEN
				lamp24On := FALSE;
				lamp27On := TRUE;
			END_IF	
			setError(roboArmStates.stErrNoPalletWaitPos);
		END_IF		
	
// *** Move to Empty - Move Check
// Проверка дали робота е стигнал над чакащата поз.

	roboArmStates.stMoveToEmptyMoveCheck:		
		IF Stations.roboData = dataRequestRobot.done THEN
			nextState(roboArmStates.stMoveToEmptySliderDown);
		END_IF
		IF Stations.roboData = dataRequestRobot.error THEN
			nextState(roboArmStates.stErrRobot);
		END_IF
		timeOutError(robotMoveTime, roboArmStates.stErrRobotTimeOut);		
		
// *** Move to Empty - Slider Down
// Слайдера слиза надолу

	roboArmStates.stMoveToEmptySliderDown:		
		io.setSR(ySlideDown, ySlideUp);	
		nextState(roboArmStates.stMoveToEmptySliderCheck);		

// *** Move to Empty - Slider Check
// Проверка дали скайдера е долу

	roboArmStates.stMoveToEmptySliderCheck:
		IF io.getSR(xSlideDown, xSlideUp) THEN 
			io.setSR(yPalletLoadGrip, yPalletLoadFree);
			IF stateDelay(palletGripTime) THEN
				palletIn         := TRUE;
				palletOnEmptyPos := FALSE;
				lamp24On 		 := FALSE;
				lamp27On         := FALSE;
				nextState(roboArmStates.stMoveToEmptyDone);				
			END_IF
		END_IF		
		timeOutError(slideTime + palletGripTime, roboArmStates.stErrSlliderNotDown);

// *** Move to Empty - Done

	roboArmStates.stMoveToEmptyDone:	
		moveToEmptyStart := FALSE;				
		nextState(roboArmStates.stEmptyToUnloadStart);		
		
// *** Empty to Unload - Start  

	roboArmStates.stEmptyToUnloadStart:		
		resetActive        := TRUE;
		Stations.roboData  := dataRequestRobot.roboPrg_HomeWithPallet;
		nextState(roboArmStates.stEmptyToPalletHome);
		
// *** Empty to Unload - Pallet Home

	roboArmStates.stEmptyToPalletHome:		
		IF Stations.roboData = dataRequestRobot.done THEN
			nextState(roboArmStates.stMoveToUnloadSync);
		END_IF
		IF Stations.roboData = dataRequestRobot.error THEN
			nextState(roboArmStates.stErrRobot);
		END_IF
		timeOutError(robotMoveTime, roboArmStates.stErrRobotTimeOut);	
			
// *** Empty to Unload - Sync
// Изходният стакер трябва да е готов преди да му се носи тара от робота

	roboArmStates.stMoveToUnloadSync:		
		depSync(Stations.sUnloadStBase, globalDeps.depSUnloadStationReady);
		nextState(roboArmStates.stEmptyToUnloadMove);						

// *** Empty to Unload - Move
// Робота тръгва към изх. стакер с празна тара

	roboArmStates.stEmptyToUnloadMove:
		emptyToUnloadStart := TRUE;	
		Stations.roboData  := dataRequestRobot.roboPrg_UnloadStacker;
		nextState(roboArmStates.stEmptyToUnloadMoveCheck);			

// *** Empty to Unload - Move Check
// Проверка дали робта е там

	roboArmStates.stEmptyToUnloadMoveCheck:
		IF Stations.roboData = dataRequestRobot.done THEN
			nextState(roboArmStates.stEmptyToUnloadDone);
		END_IF
		IF Stations.roboData = dataRequestRobot.error THEN
			nextState(roboArmStates.stErrRobot);
		END_IF
		timeOutError(robotMoveTime, roboArmStates.stErrRobotTimeOut);	

// *** Empty to Unload -Done

	roboArmStates.stEmptyToUnloadDone:
		nextState(roboArmStates.stUnloadPalletStart);		
			
// *** Unload Pallet - Start
// Занесената празна тара от робота, трябва да се закл. от изх. стакер
// на върха му

	roboArmStates.stUnloadPalletStart:		
		depSignal(globalDeps.depRoboStartLoadStacker);
		nextState(roboArmStates.stUnloadPalletSyncStacker);			
	
// *** Unload Pallet - Sync Stacker
// Цинхронизация с UnloadStacker - Робота синква, че е донесъл тара, 
// а стакера потвърждава, че я закл.
// Проверява се (на базата на xTop сензора на върха на стакера) дали изхобщо 
// робота е донесъл тара

	roboArmStates.stUnloadPalletSyncStacker:
		unloadPalletStart  := TRUE;
		emptyToUnloadStart := FALSE;
		resetActive        := FALSE;
		IF Global.palletFail THEN
			setError(roboArmStates.stErrNoPalletUnload);
			Global.palletFail := FALSE;
			resetActive       := TRUE;
        END_IF			
		depSync(Stations.sUnloadStBase, globalDeps.depSUnloadRobotUnloadGrip);		
		depWait(globalDeps.depRoboUnLoadPalletLock);
		nextState(roboArmStates.stUnlodPalletRelease);		
		
// *** Unload Pallet - Pallet Release
// Тарата е успешно закл. на върха на изходният стакер, робота
// може да я усвободи

	roboArmStates.stUnlodPalletRelease:	
		palletOnEmptyPos := FALSE;
		lamp24On         := FALSE;
		lamp27On         := FALSE;	
		io.setSR(yPalletLoadFree, yPalletLoadGrip);
		IF stateDelay (palletGripTime) THEN
			io.setSR(ySlideUp, ySlideDown);
		    nextState(roboArmStates.stUnloadPalletSlideCheck);	
       END_IF							
		
// *** Unload Pallet - Slide Check
// Когато слайдера е горе може да се синкне unloadStaker, че робота е
// освободил тарата

	roboArmStates.stUnloadPalletSlideCheck:		
		IF io.getSR(xSlideUp, xSlideDown) THEN 
			resetActive     := TRUE;
			palletIn        := FALSE;
			unLoadFixtures  := fixturesCount;		
			nextState(roboArmStates.stUnloadPalletSync);
		END_IF
		timeOutError(slideTime, roboArmStates.stErrSlideNotUp);	

// *** Unload Pallet - Sync

	roboArmStates.stUnloadPalletSync:
		depSync(Stations.sUnloadStBase, globalDeps.depSUnloadRobotOutOfReach);		
		nextState(roboArmStates.stUnloadPalletDone);		
		
// *** Unload Pallet - Done

	roboArmStates.stUnloadPalletDone:			
		unloadPalletStart := FALSE;		
		checkLoadStacker  := TRUE;		
		nextState(roboArmStates.stNextMoveStart);	

// *** Load Pallet - Start
// Робота трябва да взема вече празната тара от вх. стакер

	roboArmStates.stLoadPalletStart:			
		loadPalletStart := TRUE;	
		resetActive     := TRUE;
		nextState(roboArmStates.stLoadPalletSlideDown);

// *** Load Pallet - Slider Down
// Сваляне на слайдера

	roboArmStates.stLoadPalletSlideDown:			
		io.setSR(ySlideDown, ySlideUp);
		nextState(roboArmStates.stLoadPalletSliderCheck);	
	
// *** Load Pallet - Slider Check
// Проверка дали слайдера е в долна поз.

	roboArmStates.stLoadPalletSliderCheck:		
		IF io.getSR(xSlideDown, xSlideUp) THEN 
			io.setSR(yPalletLoadGrip, yPalletLoadFree);
			resetActive := FALSE;
			IF stateDelay(palletGripTime) THEN
				nextState(roboArmStates.stLoadPalletSignal);				
			END_IF
		END_IF		
		timeOutError(slideTime + palletGripTime, roboArmStates.stErrSlliderNotDown);			
		
// *** Load Pallet - Pallet Signal
// Синква стакера - той трябва да оключи тарата

	roboArmStates.stLoadPalletSignal:		
		depSignal(globalDeps.depSLoadRobotLoadGrip);
		nextState(roboArmStates.stLoadPalletSync);
		
// *** Load Pallet - Pallet Sync
// Изчаква стакера да завърши

	roboArmStates.stLoadPalletSync:
		depWait(GlobalDeps.depRoboLoadPalletUnlock);
		nextState(roboArmStates.stLoadPalletDone);		
		
// *** Load Pallet - Done

	roboArmStates.stLoadPalletDone:	
		palletIn        := TRUE;		
		loadPalletStart := FALSE;
		resetActive     := TRUE;	
		nextState(roboArmStates.stNextMoveStart);		

// *** Empty Pos  - Start
// Празната тара от вх. стакер трябва да се занесе на
// чакащата поз.

	roboArmStates.stEmptyPosStart:
		emptyPosStart := TRUE;
		resetActive   := TRUE;
		nextState(roboArmStates.stEmptyPosPalletHome);

// *** Empty Pos  - Pallet Home

	roboArmStates.stEmptyPosPalletHome:
		Stations.roboData     := dataRequestRobot.roboPrg_HomeWithPallet;
		nextState(roboArmStates.stEmptyPosPalletCheck);	

// *** Empty Pos  - Pallet Home Check

	roboArmStates.stEmptyPosPalletCheck:
		IF Stations.roboData = dataRequestRobot.done THEN
			nextState(roboArmStates.stEmptyPosMove);	
		END_IF	
		IF Stations.roboData = dataRequestRobot.error THEN
			nextState(roboArmStates.stErrRobot);
		END_IF
		timeOutError(robotMoveTime, roboArmStates.stErrRobotTimeOut);
		
// *** Empty Pos  - Move
// Робота се премества над чакащата поз.

	roboArmStates.stEmptyPosMove:
		Stations.roboData     := dataRequestRobot.roboPrg_EmptyPlace;
		nextState(roboArmStates.stEmptyPosMoveCheck);			
	
// *** Empty Pos  - Move Check
// Проверка дали робота е на поз.

	roboArmStates.stEmptyPosMoveCheck:	
		IF Stations.roboData = dataRequestRobot.done THEN
		    depSignal(globalDeps.depRoboStartLoadStacker);  
			IF stateDelay(sensorTime) THEN 
				IF io.getX(xWaitPos) THEN
					palletMiss := FALSE;
				ELSE
					palletMiss := TRUE;
				END_IF	
			END_IF	
			nextState(roboArmStates.stEmptyPosRelease);
		END_IF		
		IF Stations.roboData = dataRequestRobot.error THEN
			nextState(roboArmStates.stErrRobot);
		END_IF
		timeOutError(robotMoveTime, roboArmStates.stErrRobotTimeOut);			
		
// *** Empty Pos - Release
// Освобождаване на тарата

	roboArmStates.stEmptyPosRelease:	
		io.setSR(yPalletLoadFree, yPalletLoadGrip);
		IF stateDelay(palletGripTime) THEN
			io.setSR(ySlideUp, ySlideDown);
			nextState(roboArmStates.stEmptyPosSlideCheck);			
		END_IF

// *** Empty Pos - Slide Check
// Проверка дали слайдера е горe

	roboArmStates.stEmptyPosSlideCheck:
		IF io.getSR(xSlideUp, xSlideDown) THEN 
			nextState(roboArmStates.stEmptyPosSync);
		    palletIn := FALSE;			
		END_IF
		timeOutError(slideTime, roboArmStates.stErrSlideNotUp);			
		
// *** Empty Pos - Done
// Ако по някакава причина е нямало донесена тара от робота,
// вгида грешка и лампата за тара започва да мига

	roboArmStates.stEmptyPosSync:	
		palletOnEmptyPos := TRUE;
		checkLoadStacker := TRUE;		

		IF palletMiss THEN
			IF typeHEX24 THEN
				lamp24On := TRUE;
				lamp27On := FALSE;
			ELSIF typeHEX27 THEN
				lamp24On := FALSE;
				lamp27On := TRUE;	
			END_IF			
			setError(roboArmStates.stErrNoPalletWaitPos);
			emptyPosStart    := FALSE;	
		ELSE		
			nextState(roboArmStates.stEmptyPosDone);	
	
		END_IF	
		
// *** Empty Pos - Done

	roboArmStates.stEmptyPosDone:		
		emptyPosStart   := FALSE;	
		IF Global.emptyLoadPallet THEN
			blockRunForLoad   := TRUE;
			unLoadFixtures    := 0;
			depSignal(globalDeps.depRobotClearUnLoadStacker);
		ELSE	
			nextState(roboArmStates.stNextMoveStart);
		END_IF			
		
// *** Load - Start
// Робота се мести на входния стакер и чрез лазерната си ролетка
// търси сенсзор. След като намери слиза надолу и го захваща с грипера си.

	roboArmStates.stLoadStart:			
		loadStart   := TRUE;
		resetActive := TRUE;	
		IF loadFixtures = 0 THEN
			loadStart := FALSE;
			nextState(roboArmStates.stNextMoveStart);
			IF Global.lStackLastPallet THEN
				Global.emptyLoadPallet := TRUE;
			END_IF
		END_IF
		nextState(roboArmStates.stLoadMove1);		
		
// *** Load - Move 1
// Робота утива над следващата поз. на изходанта тара

	roboArmStates.stLoadMove1:		
		TagsRobot.loadPalletPos := loadFixtures;
		Stations.roboData       := dataRequestRobot.roboPrg_SensorLoad;	
		nextState(roboArmStates.stLoadMoveCheck1);

// *** Load - Move Check1
// Проверка дали робота е стигнал над зададенто гнездо
// Ако е там слиза надолу
 
	roboArmStates.stLoadMoveCheck1:	
    	IF Stations.roboData = dataRequestRobot.done AND io.getSR(ioImage.xRot_home, ioImage.xRot_back) THEN
			Stations.roboData  := dataRequestRobot.roboPrg_SensorDown;			
			nextState(roboArmStates.stLoadMoveCheck2);
		ELSIF Stations.roboData = dataRequestRobot.done	AND NOT io.getSR(ioImage.xRot_home, ioImage.xRot_back) THEN
			setError(roboArmStates.stErrRotNotTurn0);
		END_IF
		IF Stations.roboData = dataRequestRobot.error THEN
			nextState(roboArmStates.stErrRobot);
		END_IF
		timeOutError(robotMoveTime, roboArmStates.stErrRobotTimeOut);		

// *** Load - Move Check1
// Проверка дали има сензор в гнездото

	roboArmStates.stLoadMoveCheck2:	
		IF Stations.roboData = dataRequestRobot.done THEN
			IF io.getX(ioImage.xLaser) THEN
				nextState(roboArmStates.stLoadWaitCommand);			
			ELSE
				loadFixtures := loadFixtures - 1;
				nextState(roboArmStates.stLoadMove1);
			END_IF 
		END_IF		
		IF Stations.roboData = dataRequestRobot.error THEN
			nextState(roboArmStates.stErrRobot);
		END_IF
		timeOutError(robotMoveTime, roboArmStates.stErrRobotTimeOut);

// *** Load - Wait Command
// Робота изчаква някой от Inserter да си "поиска" сенсор
// LoadInserter ще иска робота да му занесе сензор
// Ако по някаква причина LoadInserer не иска сензор, то UnloadInser, 
// може да пойска робота да го разтовари

	roboArmStates.stLoadWaitCommand:	
		depNextState(Stations.insertLoadStBase, globalDeps.depILoadSignalForLoad, roboArmStates.stLoadMove2);	
		depNextState(Stations.machineStBase,    globalDeps.depMachineStopping,    roboArmStates.stStationStop);
		depNextState(Stations.machineStBase,    globalDeps.depMachineStop,        roboArmStates.stStationStop);		
		
		IF Global.sensorOnIUnload THEN
			nextState(roboArmStates.stUInsertStart);
		    loadStart               := FALSE; 	
		END_IF	
	

// *** Load - Move Check 2
// Робота е намерил сензор, затваряне на грипера

	roboArmStates.stLoadMove2:
		io.setSR(ioImage.yGrip_close, ioImage.yGrip_open);
		nextState(roboArmStates.stLoadGripCheck);
		
// *** Load - Grip Check
// Затворил ли е грипера ?

	roboArmStates.stLoadGripCheck:
		IF io.getSR(ioImage.xGrip_close, ioImage.xGrip_open) THEN
			nextState(roboArmStates.stLoadDone);	
			loadFixtures := loadFixtures - 1;			
		END_IF
		timeOutError(gripTimeOut, roboArmStates.stErrGripNotClose);			

// *** Load - Done

	roboArmStates.stLoadDone:
		loadStart := FALSE;
		nextState(roboArmStates.stLInsertStart);			
	
// *** Unload - Start
// След като е взел сензор от UnloadInserter робота трябва да го остави
// на изходната тара

	roboArmStates.stUnloadStart:			
		unloadStart   := TRUE;
		resetActive   := TRUE;	
		nextState(roboArmStates.stUnloadMove1);		
		
// *** Unload - Move 1
// Робота утива над следващата поз. на изходанта тара

	roboArmStates.stUnloadMove1:	
		io.setSR(ioImage.yRot_home, ioImage.yRot_back);		
		TagsRobot.unLoadPalletPos := unloadFixtures;
		Stations.roboData         := dataRequestRobot.roboPrg_SensorUnload;	
		nextState(roboArmStates.stUnloadMoveCheck1);	

// *** Unload - Move Check1
// Робота застава над поз. за поставяне на изходната тара

	roboArmStates.stUnloadMoveCheck1:	
		IF Stations.roboData = dataRequestRobot.done THEN
			nextState(roboArmStates.stUnloadRotCheck);			
		END_IF	
		IF Stations.roboData = dataRequestRobot.error THEN
			nextState(roboArmStates.stErrRobot);
		END_IF
		timeOutError(robotMoveTime, roboArmStates.stErrRobotTimeOut);

// *** Unload - Check Rot
// Робота слиза надолу зада остави сензора в изх. тара
// ако ротатора е на правилната поз.

	roboArmStates.stUnloadRotCheck:
		IF io.getSR(ioImage.xRot_home, ioImage.xRot_back) THEN
			Stations.roboData     := dataRequestRobot.roboPrg_SensorDown;
			nextState(roboArmStates.stUnloadMoveCheck2);
		END_IF
		timeOutError(rotTimeOut, roboArmStates.stErrRotNotTurn0);

// *** Unload - Move Check 2
// Робота трябва да си отвори грипера за да остави сензора в изх. тара

	roboArmStates.stUnloadMoveCheck2:
		IF Stations.roboData = dataRequestRobot.done THEN
			io.setSR(ioImage.yGrip_open, ioImage.yGrip_close);
		    nextState(roboArmStates.stUnloadGripCheck);				
		END_IF		
		IF Stations.roboData = dataRequestRobot.error THEN
			nextState(roboArmStates.stErrRobot);
		END_IF
		timeOutError(robotMoveTime, roboArmStates.stErrRobotTimeOut);		

// *** Unload - Grip Check
// Отворил ли е грипера ?

	roboArmStates.stUnloadGripCheck:
		IF io.getSR(ioImage.xGrip_open, ioImage.xGrip_close) THEN
		    unloadFixtures := unloadFixtures - 1;
			nextState(roboArmStates.stUnloadDone);				
		END_IF
		timeOutError(gripTimeOut, roboArmStates.stErrGripNotOpen);			

// *** Unload - Done

	roboArmStates.stUnloadDone:
		unLoadStart := FALSE;
		nextState(roboArmStates.stReady);		
		
// *** Load Insert - Start
// Робота трябва да подаде сензор на Load Inserter

	roboArmStates.stLInsertStart:			
		lInsertStart  := TRUE;
		resetActive   := TRUE;	
		nextState(roboArmStates.stLInsertMove1);			
		
// *** Load Insert - Move 1
// Робота утива на поз. малко преди грипера на инсъртъра
// Малко след кат оробота е тръгнал се завърта и сензора
// Въртенето е на базата само на таймер !

	roboArmStates.stLInsertMove1:			
		Stations.roboData       := dataRequestRobot.roboPrg_PreLoad;
		IF stateDelay (rotAfterTime) THEN
			io.setSR(ioImage.yRot_back, ioImage.yRot_home);
	    	nextState(roboArmStates.stLInsertMoveCheck1);			
		END_IF
							
// *** Load Insert - Move Check 1
// Робота изпълни ли си хода ?

	roboArmStates.stLInsertMoveCheck1:				
		IF Stations.roboData = dataRequestRobot.done THEN
		    nextState(roboArmStates.stLInsertRotCheck);				
		END_IF	
		IF Stations.roboData = dataRequestRobot.error THEN
			nextState(roboArmStates.stErrRobot);
		END_IF
		timeOutError(robotMoveTime, roboArmStates.stErrRobotTimeOut);		
		
// *** Load Insert - Rot Check
// За да може да се подаде сензора от робота на инсъртъра
// той трябва да е завъртян на 180 град. След което го подава на инсътръта

	roboArmStates.stLInsertRotCheck:		
		IF io.getSR(ioImage.xRot_back, ioImage.xRot_home) THEN
			nextState(roboArmStates.stLInsertMoveCheck2);	
		    Stations.roboData     := dataRequestRobot.roboPrg_Load;			
		END_IF
		timeOutError(rotTimeOut, roboArmStates.stErrRotNotTurn180);	

// *** Load Insert - Move Check 2
// Робота изпълни ли си хода ?

	roboArmStates.stLInsertMoveCheck2:				
		IF Stations.roboData = dataRequestRobot.done THEN
		    nextState(roboArmStates.stLInsertMoveDone);				
		END_IF		
		IF Stations.roboData = dataRequestRobot.error THEN
			nextState(roboArmStates.stErrRobot);
		END_IF
		timeOutError(robotMoveTime, roboArmStates.stErrRobotTimeOut);
		
// *** Load Insert - Done

	roboArmStates.stLInsertMoveDone:
		lInsertStart     := FALSE;	
		nextState(roboArmStates.stLInsertLockStart);	
		
// *** Load Insert Lock - Start
// Робота подава сензора на грипера на инсъттъра

	roboArmStates.stLInsertLockStart:		
        lInsertLockStart := TRUE;
		resetActive      := FALSE;		
		nextState(roboArmStates.stLInsertLockSync);
		
// *** Load Insert Lock - Sync
// Робота се синква с Load Inserter, последият може да затвори грипера си да 
// захване сензора. Робта изчаква това да се случи и тогава отваря грипера си.

	roboArmStates.stLInsertLockSync:			
		depSignal(globalDeps.depRoboILoadOnPos);		
		depSync(Stations.insertLoadStBase, globalDeps.depRoboGripOpen);
		nextState(roboArmStates.stLInsertLockGripOpen);		
	
// *** Load Insert Lock - Grip open
// Робота си отваря грипера

	roboArmStates.stLInsertLockGripOpen:		
		io.setSR(ioImage.yGrip_open, ioImage.yGrip_close);
		nextState(roboArmStates.stLInsertLockGripCheck);		
	
// *** Load Insert Lock - Grip Check
// Отворил ли се е грипера ?

	roboArmStates.stLInsertLockGripCheck:		
		IF io.getSR(ioImage.xGrip_open, ioImage.xGrip_close) THEN
			nextState(roboArmStates.stLInsertLockDone);					
		END_IF
		timeOutError(gripTimeOut, roboArmStates.stErrGripNotOpen);	
	
// *** Load Insert Lock - Done

	roboArmStates.stLInsertLockDone:
		lInsertLockStart := FALSE;		
		nextState(roboArmStates.stLInsertBackStart);		
		
// *** Load Insert Back - Start
// Робата се мръдва леко на зад след като е зареди сензор
// така инсъртъра е безппастно да рабори 

	roboArmStates.stLInsertBackStart:		
		lInsertBack  := TRUE;
		resetActive  := TRUE;
		nextState(roboArmStates.stLInsertBackMove);				
		
// *** Load Insert Back - Move
// Задава се програма на робота

	roboArmStates.stLInsertBackMove:		
		Stations.roboData := dataRequestRobot.roboPrg_PreLoad;		
		nextState(roboArmStates.stLInsertBackMoveCheck);		
		
// *** Load Insert Back - Move Check
// Робота изпълни ли си хода ?

	roboArmStates.stLInsertBackMoveCheck:
		IF Stations.roboData = dataRequestRobot.done THEN
			depSignal(globalDeps.depILoadRobotBack);				
		    nextState(roboArmStates.stLInsertBackDone);			
		END_IF		
		IF Stations.roboData = dataRequestRobot.error THEN
			nextState(roboArmStates.stErrRobot);
		END_IF
		timeOutError(robotMoveTime, roboArmStates.stErrRobotTimeOut);			
		
// *** Load Insert Back - Done
// Зависи дали има изваден сензор от UnloadIserter
// Робота или отива към него или към вх. стакер

	roboArmStates.stLInsertBackDone:
        lInsertBack	:= FALSE;
        resetActive := FALSE;		
		IF Global.sensorOnIUnload THEN 
			nextState(roboArmStates.stUInsertStart);
		END_IF
		IF loadFixtures > 0 THEN
			io.setSR(ioImage.yRot_home, ioImage.yRot_back);
			nextState(roboArmStates.stLoadStart);
		ELSE
			io.setSR(ioImage.yRot_home, ioImage.yRot_back);
			nextState(roboArmStates.stNextMoveStart);
		END_IF						
	
// *** Unload Insert - Start
// Робота трябва да вземе сензор на Unload Inserter

	roboArmStates.stUInsertStart:			
		uInsertStart           := TRUE;
		resetActive            := TRUE;	
		Global.sensorOnIUnload := FALSE;
		nextState(roboArmStates.stUInsertMove1);			
		
// *** Unload Insert - Move 1
// Робота утива на поз. малко преди грипера на инсъртъра

	roboArmStates.stUInsertMove1:			
		Stations.roboData   := dataRequestRobot.roboPrg_PreUnload;
		IF stateDelay (rotAfterTime) THEN
			io.setSR(ioImage.yRot_back, ioImage.yRot_home);
			io.setSR(ioImage.yGrip_open, ioImage.yGrip_close);
	    	nextState(roboArmStates.stUInsertMoveCheck1);			
		END_IF
							
// *** Unload Insert - Move Check 1
// Робота изпълни ли си хода ?

	roboArmStates.stUInsertMoveCheck1:				
		IF Stations.roboData = dataRequestRobot.done THEN
		    nextState(roboArmStates.stUInsertRotCheck);				
		END_IF	
		IF Stations.roboData = dataRequestRobot.error THEN
			nextState(roboArmStates.stErrRobot);
		END_IF
		timeOutError(robotMoveTime, roboArmStates.stErrRobotTimeOut);		
		
// *** Unload Insert - Rot Check
// За да може да се вземе сензора от робота на инсъртъра
// той трябва да е завъртян на 0 град. 

	roboArmStates.stUInsertRotCheck:		
		IF io.getSR(ioImage.xRot_back, ioImage.xRot_home) THEN
			nextState(roboArmStates.stUInsertSync);			
		END_IF
		timeOutError(rotTimeOut, roboArmStates.stErrRotNotTurn180);
		
// *** Unload Insert - Sync

	roboArmStates.stUInsertSync:
		depWait(globalDeps.depRoboULoadOnPos); 
		nextState(roboArmStates.stUInsertMove2);	

// *** Unload Insert - Move 2
// Когато инсертъра е готов, робота се преближава за да вземе сензор

	roboArmStates.stUInsertMove2:	
		Stations.roboData     := dataRequestRobot.roboPrg_Unload;	
		nextState(roboArmStates.stUInsertMoveCheck2);		

// *** Unload Insert - Move Check 2
// Робота изпълни ли си хода ?

	roboArmStates.stUInsertMoveCheck2:				
		IF Stations.roboData = dataRequestRobot.done THEN
		    nextState(roboArmStates.stUInsertMoveDone);				
		END_IF	
		IF Stations.roboData = dataRequestRobot.error THEN
			nextState(roboArmStates.stErrRobot);
		END_IF
		timeOutError(robotMoveTime, roboArmStates.stErrRobotTimeOut);
		
// *** Unload Insert - Done

	roboArmStates.stUInsertMoveDone:
		uInsertStart     := FALSE;	
		nextState(roboArmStates.stUInsertLockStart);	

// *** Unload Insert Lock - Start
// Робота взима сензора от грипера на инсъттъра

	roboArmStates.stUInsertLockStart:		
        uInsertLockStart := TRUE;
		resetActive      := FALSE;			
		nextState(roboArmStates.stUInsertLockGripClose);		
	
// *** Unload Insert Lock - Grip Close
// Робота си затваря грипера

	roboArmStates.stUInsertLockGripClose:		
		io.setSR(ioImage.yGrip_close, ioImage.yGrip_open);
		IF stateDelay(gripTime) THEN
			nextState(roboArmStates.stUInsertLockGripCheck);	
		END_IF	
	
// *** Unload Insert Lock - Grip Check
// Затворил ли се е грипера ?

	roboArmStates.stUInsertLockGripCheck:		
		IF io.getSR(ioImage.xGrip_close, ioImage.xGrip_open) THEN
			nextState(roboArmStates.stUInsertLockSync);					
		END_IF
		timeOutError(gripTimeOut, roboArmStates.stErrGripNotClose);	
		
// *** Unload Insert Lock - Sync
// Робота се синква с UnLoad Inserter. 
	roboArmStates.stUInsertLockSync:			
		depSignal(globalDeps.depRoboGripClose);
		depSync(Stations.insertUnLoadStBase, globalDeps.depRoboLoadSensor);	
		nextState(roboArmStates.stUInsertLockDone);
	
// *** Unload Insert Lock - Done

	roboArmStates.stUInsertLockDone:
		uInsertLockStart := FALSE;		
		nextState(roboArmStates.stUInsertBackStart);	

// *** Unload Insert Back - Start
// Робата се мръдва леко на зад след като е взел сензор

